KUKA KRL program: EPS_2_25694_RR04_A_20260114065914.src

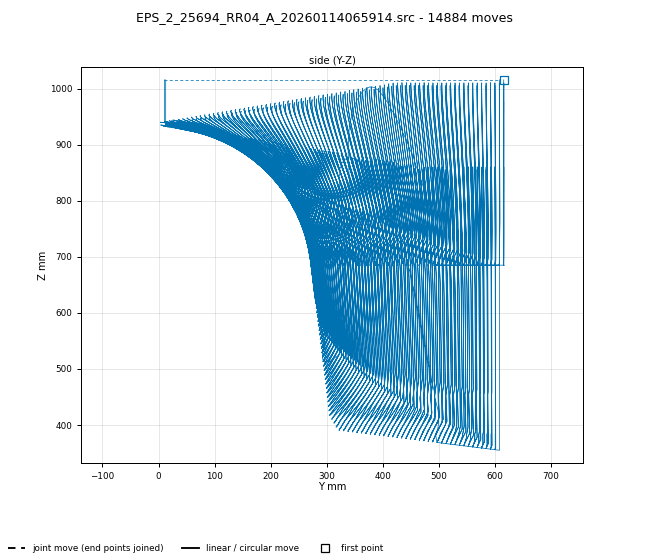
[picture p0: tool path of EPS_2_25694_RR04_A_20260114065914.src, 14884 of 14886 moves have a stored position in this frame; points joined in program order, loops and branches not executed]
&ACCESS RVP
&REL 4
&COMMENT QRS 19112012
&PARAM EDITMASK = *
DEF PART()
EXT BAS (BAS_COMMAND :IN,REAL :IN )
INT I
BAS (#INITMOV,0 )

;KUKA QRS Post kuka4.cps  Date:22-06-2017 !

File_ID=2965

QRS_PRE_INIT()

;Init var - Until changes are made in qrs_pre_init
Outlet_Square_prg=0
Inlet_1_Square_prg=0
Inlet_2_Square_prg=0
Inlet_3_Square_prg=0
Inlet_4_Square_prg=0
Inlet_5_Square_prg=0

Outlet_1={X 0.000, Y 425.000, Z 739.000, B 0.000, E1 0.000 }
Inlet_1={X 0.000, Y 466.000, Z 567.000, B 0.000, E1 180.000 }
Outlet_1_type=533
Inlet_1_type=457
;QRS#1=Sidecore dimensions
;QRS#2=525-21" Concrete
;QRS#3=450-18" Concrete
;QRS#4=
;QRS#5=
;QRS#6=
;QRS#7=
;QRS#8=
;QRS#9=S306-32
;QRS#10=28A PSX-2
;QRS#11=
;QRS#12=
;QRS#13=
;QRS#14=
;QRS#15=
;QRS#16=1220x127x1372 4,5'
;QRS#17=EPS Height
;QRS#18=1005,5
;QRS#19=*
;QRS#20= UPDATED VERSION 22-06-2017
;QRS#21=*
Outlet_Square=0250
Inlet_1_Square=0250
Inlet_2_Square=0
Inlet_3_Square=0
Inlet_4_Square=0
Inlet_5_Square=0
Mill_Square=1
Outlet_Square_Prg=263
Inlet_1_Square_prg=274

QRS_INIT()

$ADVANCE=5

; T1
PTP {E1 172.545,E2 172.545}
PTP {X 0,Y 615.546,A -85,B 0,C 180,E1 172.545,E2 172.545,E3 0,E4 0,E5 0,E6 0}
QRS_SPEED_INIT()
LIN {X 0,Y 615.546,Z 1015.5,A -85,B 0,C 180,E1 172.545,E2 172.545,E3 0,E4 0,E5 0,E6 0} C_VEL
LIN {X 0,Y 615.546,Z 687.03,A -85,B 0,C 180,E1 172.545,E2 172.545} C_VEL
LIN {X 0,Y 615.492,Z 685.03,A -85,B 0,C 180,E1 172.731,E2 172.731} C_VEL
LIN {X 0,Y 615.811,Z 685.03,A -85,B 0,C 180,E1 176.52,E2 176.52} C_VEL
LIN {X 0,Y 615.861,Z 685.03,A -85,B 0,C 180,E1 181.159,E2 181.159} C_VEL
LIN {X 0,Y 615.796,Z 685.03,A -85,B 0,C 180,E1 185.807,E2 185.807} C_VEL
LIN {X 0,Y 615.764,Z 685.03,A -85,B 0,C 180,E1 190.494,E2 190.494} C_VEL
LIN {X 0,Y 615.78,Z 685.03,A -85,B 0,C 180,E1 195.253,E2 195.253} C_VEL
LIN {X 0,Y 615.726,Z 685.03,A -85,B 0,C 180,E1 200.124,E2 200.124} C_VEL
LIN {X 0,Y 615.726,Z 685.03,A -85,B 0,C 180,E1 205.151,E2 205.151} C_VEL
LIN {X 0,Y 615.183,Z 685.03,A -85,B 0,C 180,E1 207.768,E2 207.768} C_VEL
LIN {X 0,Y 615.676,Z 685.03,A -85,B 0,C 180,E1 210.398,E2 210.398} C_VEL
LIN {X 0,Y 615.111,Z 685.03,A -85,B 0,C 180,E1 213.847,E2 213.847} C_VEL
LIN {X 0,Y 615.672,Z 685.03,A -85,B 0,C 180,E1 215.942,E2 215.942} C_VEL
LIN {X 0,Y 615.221,Z 685.03,A -85,B 0,C 180,E1 217.827,E2 217.827} C_VEL
LIN {X 0,Y 615.646,Z 685.03,A -85,B 0,C 180,E1 221.91,E2 221.91} C_VEL
LIN {X 0,Y 615.206,Z 685.03,A -85,B 0,C 180,E1 225.149,E2 225.149} C_VEL
LIN {X 0,Y 615.631,Z 685.03,A -85,B 0,C 180,E1 228.094,E2 228.094} C_VEL
LIN {X 0,Y 615.6,Z 685.03,A -85,B 0,C 180,E1 232.135,E2 232.135} C_VEL
LIN {X 0,Y 615.584,Z 685.03,A -85,B 0,C 180,E1 234.056,E2 234.056} C_VEL
LIN {X 0,Y 615.733,Z 685.03,A -85,B 0,C 180,E1 236.075,E2 236.075} C_VEL
LIN {X 0,Y 615.772,Z 685.03,A -85,B 0,C 180,E1 236.884,E2 236.884} C_VEL
LIN {X 0,Y 615.674,Z 685.03,A -85,B 0,C 180,E1 239.605,E2 239.605} C_VEL
LIN {X 0,Y 615.593,Z 685.03,A -85,B 0,C 180,E1 240.51,E2 240.51} C_VEL
LIN {X 0,Y 615.33,Z 685.03,A -85,B 0,C 180,E1 240.559,E2 240.559} C_VEL
LIN {X 0,Y 615.244,Z 685.519,A -85,B 0,C 180,E1 240.579,E2 240.579} C_VEL
LIN {X 0,Y 615.438,Z 754.445,A -85,B 0,C 180,E1 241.499,E2 241.499} C_VEL
LIN {X 0,Y 615.518,Z 765.253,A -85,B 0,C 180,E1 241.679,E2 241.679} C_VEL
LIN {X 0,Y 615.547,Z 778.462,A -85,B 0,C 180,E1 241.958,E2 241.958} C_VEL
LIN {X 0,Y 615.507,Z 788.764,A -85,B 0,C 180,E1 242.217,E2 242.217} C_VEL
LIN {X 0,Y 615.684,Z 804.589,A -85,B 0,C 180,E1 242.709,E2 242.709} C_VEL
LIN {X 0,Y 615.643,Z 817.012,A -85,B 0,C 180,E1 243.155,E2 243.155} C_VEL
LIN {X 0,Y 615.565,Z 826.929,A -85,B 0,C 180,E1 243.556,E2 243.556} C_VEL
LIN {X 0,Y 615.705,Z 842.642,A -85,B 0,C 180,E1 244.289,E2 244.289} C_VEL
LIN {X 0,Y 615.691,Z 854.976,A -85,B 0,C 180,E1 244.938,E2 244.938} C_VEL
LIN {X 0,Y 615.678,Z 866.612,A -85,B 0,C 180,E1 245.617,E2 245.617} C_VEL
LIN {X 0,Y 615.714,Z 878.42,A -85,B 0,C 180,E1 246.381,E2 246.381} C_VEL
LIN {X 0,Y 615.719,Z 889.111,A -85,B 0,C 180,E1 247.137,E2 247.137} C_VEL
LIN {X 0,Y 615.716,Z 900.416,A -85,B 0,C 180,E1 248.014,E2 248.014} C_VEL
LIN {X 0,Y 615.703,Z 909.675,A -85,B 0,C 180,E1 248.793,E2 248.793} C_VEL
LIN {X 0,Y 615.752,Z 919.81,A -85,B 0,C 180,E1 249.725,E2 249.725} C_VEL
LIN {X 0,Y 615.721,Z 929.071,A -85,B 0,C 180,E1 250.648,E2 250.648} C_VEL
LIN {X 0,Y 615.679,Z 937.431,A -85,B 0,C 180,E1 251.55,E2 251.55} C_VEL
LIN {X 0,Y 615.758,Z 945.789,A -85,B 0,C 180,E1 252.533,E2 252.533} C_VEL
LIN {X 0,Y 615.711,Z 953.693,A -85,B 0,C 180,E1 253.543,E2 253.543} C_VEL
LIN {X 0,Y 615.576,Z 960.436,A -85,B 0,C 180,E1 254.474,E2 254.474} C_VEL
LIN {X 0,Y 615.669,Z 968.069,A -85,B 0,C 180,E1 255.646,E2 255.646} C_VEL
LIN {X 0,Y 615.808,Z 973.445,A -85,B 0,C 180,E1 256.545,E2 256.545} C_VEL
LIN {X 0,Y 615.572,Z 979.916,A -85,B 0,C 180,E1 257.729,E2 257.729} C_VEL
LIN {X 0,Y 615.608,Z 985.63,A -85,B 0,C 180,E1 258.914,E2 258.914} C_VEL
LIN {X 0,Y 615.819,Z 990.639,A -85,B 0,C 180,E1 260.097,E2 260.097} C_VEL
LIN {X 0,Y 615.602,Z 995.067,A -85,B 0,C 180,E1 261.269,E2 261.269} C_VEL
LIN {X 0,Y 615.662,Z 999.448,A -85,B 0,C 180,E1 262.653,E2 262.653} C_VEL
LIN {X 0,Y 615.802,Z 1002.364,A -85,B 0,C 180,E1 263.748,E2 263.748} C_VEL
LIN {X 0,Y 615.545,Z 1005.382,A -85,B 0,C 180,E1 265.123,E2 265.123} C_VEL
LIN {X 0,Y 615.635,Z 1007.593,A -85,B 0,C 180,E1 266.519,E2 266.519} C_VEL
LIN {X 0,Y 615.819,Z 1008.67,A -85,B 0,C 180,E1 267.449,E2 267.449} C_VEL
LIN {X 0,Y 615.544,Z 1009.716,A -85,B 0,C 180,E1 268.84,E2 268.84} C_VEL
LIN {X 0,Y 615.842,Z 1009.659,A -85,B 0,C 180,E1 271.16,E2 271.16} C_VEL
LIN {X 0,Y 615.626,Z 1009.07,A -85,B 0,C 180,E1 272.088,E2 272.088} C_VEL
LIN {X 0,Y 615.536,Z 1007.611,A -85,B 0,C 180,E1 273.482,E2 273.482} C_VEL
LIN {X 0,Y 615.805,Z 1005.333,A -85,B 0,C 180,E1 274.875,E2 274.875} C_VEL
LIN {X 0,Y 615.605,Z 1002.405,A -85,B 0,C 180,E1 276.252,E2 276.252} C_VEL
LIN {X 0,Y 615.625,Z 999.258,A -85,B 0,C 180,E1 277.421,E2 277.421} C_VEL
LIN {X 0,Y 615.798,Z 995.034,A -85,B 0,C 180,E1 278.729,E2 278.729} C_VEL
LIN {X 0,Y 615.583,Z 990.671,A -85,B 0,C 180,E1 279.907,E2 279.907} C_VEL
LIN {X 0,Y 615.638,Z 985.623,A -85,B 0,C 180,E1 281.086,E2 281.086} C_VEL
LIN {X 0,Y 615.808,Z 979.885,A -85,B 0,C 180,E1 282.267,E2 282.267} C_VEL
LIN {X 0,Y 615.627,Z 973.459,A -85,B 0,C 180,E1 283.46,E2 283.46} C_VEL
LIN {X 0,Y 615.697,Z 966.199,A -85,B 0,C 180,E1 284.654,E2 284.654} C_VEL
LIN {X 0,Y 615.81,Z 960.634,A -85,B 0,C 180,E1 285.488,E2 285.488} C_VEL
LIN {X 0,Y 615.662,Z 951.204,A -85,B 0,C 180,E1 286.79,E2 286.79} C_VEL
LIN {X 0,Y 615.736,Z 942.609,A -85,B 0,C 180,E1 287.852,E2 287.852} C_VEL
LIN {X 0,Y 615.77,Z 934.421,A -85,B 0,C 180,E1 288.783,E2 288.783} C_VEL
LIN {X 0,Y 615.695,Z 924.535,A -85,B 0,C 180,E1 289.815,E2 289.815} C_VEL
LIN {X 0,Y 615.712,Z 916.55,A -85,B 0,C 180,E1 290.587,E2 290.587} C_VEL
LIN {X 0,Y 615.743,Z 906.049,A -85,B 0,C 180,E1 291.517,E2 291.517} C_VEL
LIN {X 0,Y 615.702,Z 896.053,A -85,B 0,C 180,E1 292.335,E2 292.335} C_VEL
LIN {X 0,Y 615.701,Z 886.308,A -85,B 0,C 180,E1 293.07,E2 293.07} C_VEL
LIN {X 0,Y 615.683,Z 874.638,A -85,B 0,C 180,E1 293.873,E2 293.873} C_VEL
LIN {X 0,Y 615.697,Z 862.6,A -85,B 0,C 180,E1 294.623,E2 294.623} C_VEL
LIN {X 0,Y 615.65,Z 851.918,A -85,B 0,C 180,E1 295.232,E2 295.232} C_VEL
LIN {X 0,Y 615.643,Z 841.055,A -85,B 0,C 180,E1 295.795,E2 295.795} C_VEL
LIN {X 0,Y 615.699,Z 826.912,A -85,B 0,C 180,E1 296.438,E2 296.438} C_VEL
LIN {X 0,Y 615.612,Z 813.716,A -85,B 0,C 180,E1 296.969,E2 296.969} C_VEL
LIN {X 0,Y 615.55,Z 804.569,A -85,B 0,C 180,E1 297.298,E2 297.298} C_VEL
LIN {X 0,Y 615.613,Z 787.831,A -85,B 0,C 180,E1 297.801,E2 297.801} C_VEL
LIN {X 0,Y 615.471,Z 776.05,A -85,B 0,C 180,E1 298.103,E2 298.103} C_VEL
LIN {X 0,Y 615.643,Z 762.933,A -85,B 0,C 180,E1 298.359,E2 298.359} C_VEL
LIN {X 0,Y 615.608,Z 744.148,A -85,B 0,C 180,E1 298.636,E2 298.636} C_VEL
LIN {X 0,Y 615.246,Z 685.03,A -85,B 0,C 180,E1 299.433,E2 299.433} C_VEL
LIN {X 0,Y 615.499,Z 685.03,A -85,B 0,C 180,E1 299.474,E2 299.474} C_VEL
LIN {X 0,Y 615.685,Z 685.03,A -85,B 0,C 180,E1 300.395,E2 300.395} C_VEL
LIN {X 0,Y 615.866,Z 685.03,A -85,B 0,C 180,E1 303.111,E2 303.111} C_VEL
LIN {X 0,Y 615.556,Z 685.03,A -85,B 0,C 180,E1 305.946,E2 305.946} C_VEL
LIN {X 0,Y 615.615,Z 685.03,A -85,B 0,C 180,E1 307.866,E2 307.866} C_VEL
LIN {X 0,Y 615.631,Z 685.03,A -85,B 0,C 180,E1 311.906,E2 311.906} C_VEL
LIN {X 0,Y 615.209,Z 685.03,A -85,B 0,C 180,E1 315.144,E2 315.144} C_VEL
LIN {X 0,Y 615.686,Z 685.03,A -85,B 0,C 180,E1 318.094,E2 318.094} C_VEL
LIN {X 0,Y 615.541,Z 685.03,A -85,B 0,C 180,E1 322.136,E2 322.136} C_VEL
LIN {X 0,Y 615.511,Z 685.03,A -85,B 0,C 180,E1 324.047,E2 324.047} C_VEL
LIN {X 0,Y 615.673,Z 685.03,A -85,B 0,C 180,E1 326.076,E2 326.076} C_VEL
LIN {X 0,Y 615.675,Z 685.03,A -85,B 0,C 180,E1 326.874,E2 326.874} C_VEL
LIN {X 0,Y 615.495,Z 685.03,A -85,B 0,C 180,E1 330.517,E2 330.517} C_VEL
LIN {X 0,Y 615.462,Z 685.03,A -85,B 0,C 180,E1 332.245,E2 332.245} C_VEL
LIN {X 0,Y 615.386,Z 685.03,A -85,B 0,C 180,E1 335.665,E2 335.665} C_VEL
LIN {X 0,Y 615.551,Z 685.03,A -85,B 0,C 180,E1 337.379,E2 337.379} C_VEL
LIN {X 0,Y 615.774,Z 685.03,A -85,B 0,C 180,E1 341.999,E2 341.999} C_VEL
LIN {X 0,Y 615.786,Z 685.03,A -85,B 0,C 180,E1 342.329,E2 342.329} C_VEL
LIN {X 0,Y 615.756,Z 685.03,A -85,B 0,C 180,E1 347.137,E2 347.137} C_VEL
LIN {X 0,Y 615.771,Z 685.03,A -85,B 0,C 180,E1 351.856,E2 351.856} C_VEL
LIN {X 0,Y 615.848,Z 685.03,A -85,B 0,C 180,E1 356.52,E2 356.52} C_VEL
LIN {X 0,Y 615.86,Z 685.03,A -85,B 0,C 180,E1 361.159,E2 361.159} C_VEL
LIN {X 0,Y 615.803,Z 685.03,A -85,B 0,C 180,E1 365.807,E2 365.807} C_VEL
LIN {X 0,Y 615.789,Z 685.03,A -85,B 0,C 180,E1 370.494,E2 370.494} C_VEL
LIN {X 0,Y 615.809,Z 685.03,A -85,B 0,C 180,E1 375.252,E2 375.252} C_VEL
LIN {X 0,Y 615.742,Z 685.03,A -85,B 0,C 180,E1 380.124,E2 380.124} C_VEL
LIN {X 0,Y 615.764,Z 685.03,A -85,B 0,C 180,E1 385.15,E2 385.15} C_VEL
LIN {X 0,Y 615.376,Z 685.03,A -85,B 0,C 180,E1 389.463,E2 389.463} C_VEL
LIN {X 0,Y 615.696,Z 685.03,A -85,B 0,C 180,E1 390.397,E2 390.397} C_VEL
LIN {X 0,Y 615.123,Z 685.03,A -85,B 0,C 180,E1 393.848,E2 393.848} C_VEL
LIN {X 0,Y 615.679,Z 685.03,A -85,B 0,C 180,E1 395.942,E2 395.942} C_VEL
LIN {X 0,Y 615.41,Z 685.03,A -85,B 0,C 180,E1 397.848,E2 397.848} C_VEL
LIN {X 0,Y 615.356,Z 685.03,A -85,B 0,C 180,E1 398.886,E2 398.886} C_VEL
LIN {X 0,Y 615.631,Z 685.03,A -85,B 0,C 180,E1 401.507,E2 401.507} C_VEL
LIN {X 0,Y 615.653,Z 685.03,A -85,B 0,C 180,E1 405.107,E2 405.107} C_VEL
LIN {X 0,Y 615.249,Z 685.03,A -85,B 0,C 180,E1 408.539,E2 408.539} C_VEL
LIN {X 0,Y 615.649,Z 685.03,A -85,B 0,C 180,E1 411.14,E2 411.14} C_VEL
LIN {X 0,Y 615.653,Z 685.03,A -85,B 0,C 180,E1 416.086,E2 416.086} C_VEL
LIN {X 0,Y 615.746,Z 685.03,A -85,B 0,C 180,E1 416.881,E2 416.881} C_VEL
LIN {X 0,Y 615.563,Z 685.03,A -85,B 0,C 180,E1 420.515,E2 420.515} C_VEL
LIN {X 0,Y 615.554,Z 685.03,A -85,B 0,C 180,E1 422.252,E2 422.252} C_VEL
LIN {X 0,Y 615.586,Z 685.03,A -85,B 0,C 180,E1 425.635,E2 425.635} C_VEL
LIN {X 0,Y 615.626,Z 685.03,A -85,B 0,C 180,E1 426.524,E2 426.524} C_VEL
LIN {X 0,Y 615.741,Z 696.131,A -85,B 0,C 180,E1 426.945,E2 426.945} C_VEL
LIN {X 0,Y 615.761,Z 704.206,A -85,B 0,C 180,E1 427.278,E2 427.278} C_VEL
LIN {X 0,Y 615.706,Z 714.196,A -85,B 0,C 180,E1 427.733,E2 427.733} C_VEL
LIN {X 0,Y 615.726,Z 725.668,A -85,B 0,C 180,E1 428.326,E2 428.326} C_VEL
LIN {X 0,Y 615.756,Z 736.464,A -85,B 0,C 180,E1 428.95,E2 428.95} C_VEL
LIN {X 0,Y 615.75,Z 746.203,A -85,B 0,C 180,E1 429.569,E2 429.569} C_VEL
LIN {X 0,Y 615.753,Z 755.081,A -85,B 0,C 180,E1 430.187,E2 430.187} C_VEL
LIN {X 0,Y 615.748,Z 765.126,A -85,B 0,C 180,E1 430.955,E2 430.955} C_VEL
LIN {X 0,Y 615.773,Z 773.255,A -85,B 0,C 180,E1 431.632,E2 431.632} C_VEL
LIN {X 0,Y 615.741,Z 782.057,A -85,B 0,C 180,E1 432.43,E2 432.43} C_VEL
LIN {X 0,Y 615.697,Z 789.212,A -85,B 0,C 180,E1 433.131,E2 433.131} C_VEL
LIN {X 0,Y 615.74,Z 797.147,A -85,B 0,C 180,E1 433.981,E2 433.981} C_VEL
LIN {X 0,Y 615.809,Z 803.754,A -85,B 0,C 180,E1 434.749,E2 434.749} C_VEL
LIN {X 0,Y 615.685,Z 810.869,A -85,B 0,C 180,E1 435.646,E2 435.646} C_VEL
LIN {X 0,Y 615.683,Z 817.337,A -85,B 0,C 180,E1 436.541,E2 436.541} C_VEL
LIN {X 0,Y 615.817,Z 823.206,A -85,B 0,C 180,E1 437.437,E2 437.437} C_VEL
LIN {X 0,Y 615.707,Z 828.568,A -85,B 0,C 180,E1 438.324,E2 438.324} C_VEL
LIN {X 0,Y 615.629,Z 834.87,A -85,B 0,C 180,E1 439.504,E2 439.504} C_VEL
LIN {X 0,Y 615.74,Z 839.094,A -85,B 0,C 180,E1 440.389,E2 440.389} C_VEL
LIN {X 0,Y 615.768,Z 842.865,A -85,B 0,C 180,E1 441.271,E2 441.271} C_VEL
LIN {X 0,Y 615.623,Z 847.726,A -85,B 0,C 180,E1 442.579,E2 442.579} C_VEL
LIN {X 0,Y 615.757,Z 851.304,A -85,B 0,C 180,E1 443.75,E2 443.75} C_VEL
LIN {X 0,Y 615.736,Z 853.695,A -85,B 0,C 180,E1 444.658,E2 444.658} C_VEL
LIN {X 0,Y 615.634,Z 856.541,A -85,B 0,C 180,E1 446.054,E2 446.054} C_VEL
LIN {X 0,Y 615.679,Z 857.314,A -85,B 0,C 180,E1 446.519,E2 446.519} C_VEL
LIN {X 0,Y 615.827,Z 858.489,A -85,B 0,C 180,E1 447.448,E2 447.448} C_VEL
LIN {X 0,Y 615.722,Z 859.014,A -85,B 0,C 180,E1 447.912,E2 447.912} C_VEL
LIN {X 0,Y 615.59,Z 859.697,A -85,B 0,C 180,E1 448.84,E2 448.84} C_VEL
LIN {X 0,Y 615.619,Z 859.93,A -85,B 0,C 180,E1 449.768,E2 449.768} C_VEL
LIN {X 0,Y 615.785,Z 859.595,A -85,B 0,C 180,E1 451.159,E2 451.159} C_VEL
LIN {X 0,Y 615.595,Z 858.426,A -85,B 0,C 180,E1 452.552,E2 452.552} C_VEL
LIN {X 0,Y 615.657,Z 857.167,A -85,B 0,C 180,E1 453.481,E2 453.481} C_VEL
LIN {X 0,Y 615.748,Z 856.37,A -85,B 0,C 180,E1 453.945,E2 453.945} C_VEL
LIN {X 0,Y 615.735,Z 854.511,A -85,B 0,C 180,E1 454.875,E2 454.875} C_VEL
LIN {X 0,Y 615.653,Z 853.513,A -85,B 0,C 180,E1 455.342,E2 455.342} C_VEL
LIN {X 0,Y 615.602,Z 849.864,A -85,B 0,C 180,E1 456.665,E2 456.665} C_VEL
LIN {X 0,Y 615.761,Z 847.084,A -85,B 0,C 180,E1 457.52,E2 457.52} C_VEL
LIN {X 0,Y 615.802,Z 844.751,A -85,B 0,C 180,E1 458.142,E2 458.142} C_VEL
LIN {X 0,Y 615.65,Z 841.238,A -85,B 0,C 180,E1 459.024,E2 459.024} C_VEL
LIN {X 0,Y 615.622,Z 838.719,A -85,B 0,C 180,E1 459.612,E2 459.612} C_VEL
LIN {X 0,Y 615.757,Z 832.894,A -85,B 0,C 180,E1 460.788,E2 460.788} C_VEL
LIN {X 0,Y 615.749,Z 828.046,A -85,B 0,C 180,E1 461.675,E2 461.675} C_VEL
LIN {X 0,Y 615.66,Z 822.681,A -85,B 0,C 180,E1 462.566,E2 462.566} C_VEL
LIN {X 0,Y 615.742,Z 815.692,A -85,B 0,C 180,E1 463.606,E2 463.606} C_VEL
LIN {X 0,Y 615.788,Z 809.065,A -85,B 0,C 180,E1 464.501,E2 464.501} C_VEL
LIN {X 0,Y 615.684,Z 800.716,A -85,B 0,C 180,E1 465.523,E2 465.523} C_VEL
LIN {X 0,Y 615.718,Z 793.726,A -85,B 0,C 180,E1 466.306,E2 466.306} C_VEL
LIN {X 0,Y 615.785,Z 785.347,A -85,B 0,C 180,E1 467.162,E2 467.162} C_VEL
LIN {X 0,Y 615.744,Z 777.922,A -85,B 0,C 180,E1 467.865,E2 467.865} C_VEL
LIN {X 0,Y 615.74,Z 769.905,A -85,B 0,C 180,E1 468.566,E2 468.566} C_VEL
LIN {X 0,Y 615.748,Z 760.061,A -85,B 0,C 180,E1 469.351,E2 469.351} C_VEL
LIN {X 0,Y 615.758,Z 750.554,A -85,B 0,C 180,E1 470.044,E2 470.044} C_VEL
LIN {X 0,Y 615.741,Z 741.275,A -85,B 0,C 180,E1 470.662,E2 470.662} C_VEL
LIN {X 0,Y 615.705,Z 731.012,A -85,B 0,C 180,E1 471.285,E2 471.285} C_VEL
LIN {X 0,Y 615.735,Z 721.063,A -85,B 0,C 180,E1 471.829,E2 471.829} C_VEL
LIN {X 0,Y 615.723,Z 710.661,A -85,B 0,C 180,E1 472.343,E2 472.343} C_VEL
LIN {X 0,Y 615.656,Z 699.442,A -85,B 0,C 180,E1 472.837,E2 472.837} C_VEL
LIN {X 0,Y 615.443,Z 689.43,A -85,B 0,C 180,E1 473.235,E2 473.235} C_VEL
LIN {X 0,Y 615.249,Z 685.03,A -85,B 0,C 180,E1 473.397,E2 473.397} C_VEL
LIN {X 0,Y 615.705,Z 685.03,A -85,B 0,C 180,E1 473.504,E2 473.504} C_VEL
LIN {X 0,Y 615.521,Z 685.03,A -85,B 0,C 180,E1 474.765,E2 474.765} C_VEL
LIN {X 0,Y 615.766,Z 685.03,A -85,B 0,C 180,E1 477.736,E2 477.736} C_VEL
LIN {X 0,Y 615.191,Z 685.03,A -85,B 0,C 180,E1 480.421,E2 480.421} C_VEL
LIN {X 0,Y 615.731,Z 685.03,A -85,B 0,C 180,E1 483.119,E2 483.119} C_VEL
LIN {X 0,Y 615.647,Z 685.03,A -85,B 0,C 180,E1 483.913,E2 483.913} C_VEL
LIN {X 0,Y 615.65,Z 685.03,A -85,B 0,C 180,E1 488.859,E2 488.859} C_VEL
LIN {X 0,Y 615.238,Z 685.03,A -85,B 0,C 180,E1 491.938,E2 491.938} C_VEL
LIN {X 0,Y 615.647,Z 685.03,A -85,B 0,C 180,E1 494.892,E2 494.892} C_VEL
LIN {X 0,Y 615.63,Z 685.03,A -85,B 0,C 180,E1 498.492,E2 498.492} C_VEL
LIN {X 0,Y 615.363,Z 685.03,A -85,B 0,C 180,E1 501.115,E2 501.115} C_VEL
LIN {X 0,Y 615.412,Z 685.03,A -85,B 0,C 180,E1 502.15,E2 502.15} C_VEL
LIN {X 0,Y 615.688,Z 685.03,A -85,B 0,C 180,E1 504.059,E2 504.059} C_VEL
LIN {X 0,Y 615.124,Z 685.03,A -85,B 0,C 180,E1 506.84,E2 506.84} C_VEL
LIN {X 0,Y 615.697,Z 685.03,A -85,B 0,C 180,E1 509.603,E2 509.603} C_VEL
LIN {X 0,Y 615.213,Z 685.03,A -85,B 0,C 180,E1 512.233,E2 512.233} C_VEL
LIN {X 0,Y 615.762,Z 685.03,A -85,B 0,C 180,E1 514.85,E2 514.85} C_VEL
LIN {X 0,Y 615.747,Z 685.03,A -85,B 0,C 180,E1 519.877,E2 519.877} C_VEL
LIN {X 0,Y 615.473,Z 685.03,A -85,B 0,C 180,E1 522.32,E2 522.32} C_VEL
LIN {X 0,Y 615.601,Z 685.03,A -85,B 0,C 180,E1 524.743,E2 524.743} C_VEL
LIN {X 0,Y 615.815,Z 685.03,A -85,B 0,C 180,E1 527.139,E2 527.139} C_VEL
LIN {X 0,Y 615.786,Z 685.03,A -85,B 0,C 180,E1 531.856,E2 531.856} C_VEL
LIN {X 0,Y 615.492,Z 685.03,A -85,B 0,C 180,E1 532.731,E2 532.731} C_VEL
LIN {X 0,Y 611.488,Z 685.03,A -85,B 0,C 180,E1 534.318,E2 534.318} C_VEL
LIN {X 0,Y 607.633,Z 685.03,A -85,B 0,C 180,E1 535.926,E2 535.926} C_VEL
LIN {X 0,Y 607.869,Z 685.03,A -85,B 0,C 180,E1 541.425,E2 541.425} C_VEL
LIN {X 0,Y 607.617,Z 685.03,A -85,B 0,C 180,E1 546.595,E2 546.595} C_VEL
LIN {X 0,Y 607.525,Z 685.03,A -85,B 0,C 180,E1 551.463,E2 551.463} C_VEL
LIN {X 0,Y 607.629,Z 685.03,A -85,B 0,C 180,E1 555.855,E2 555.855} C_VEL
LIN {X 0,Y 607.738,Z 685.03,A -85,B 0,C 180,E1 560.343,E2 560.343} C_VEL
LIN {X 0,Y 607.749,Z 685.03,A -85,B 0,C 180,E1 564.968,E2 564.968} C_VEL
LIN {X 0,Y 607.546,Z 685.03,A -85,B 0,C 180,E1 569.786,E2 569.786} C_VEL
LIN {X 0,Y 607.544,Z 685.03,A -85,B 0,C 180,E1 576.592,E2 576.592} C_VEL
LIN {X 0,Y 607.666,Z 685.03,A -85,B 0,C 180,E1 582.104,E2 582.104} C_VEL
LIN {X 0,Y 607.705,Z 685.03,A -85,B 0,C 180,E1 588.152,E2 588.152} C_VEL
LIN {X 0,Y 607.619,Z 685.03,A -85,B 0,C 180,E1 593.414,E2 593.414} C_VEL
LIN {X 0,Y 607.66,Z 685.03,A -85,B 0,C 180,E1 598.568,E2 598.568} C_VEL
LIN {X 0,Y 607.716,Z 685.03,A -85,B 0,C 180,E1 600.166,E2 600.166} C_VEL
LIN {X 0,Y 608.571,Z 773.176,A -85,B 0,C 180,E1 601.49,E2 601.49} C_VEL
LIN {X 0,Y 608.554,Z 810.788,A -85,B 0,C 180,E1 602.586,E2 602.586} C_VEL
LIN {X 0,Y 608.43,Z 846.811,A -85,B 0,C 180,E1 604.178,E2 604.178} C_VEL
LIN {X 0,Y 608.276,Z 881.947,A -85,B 0,C 180,E1 606.323,E2 606.323} C_VEL
LIN {X 0,Y 608.109,Z 914.005,A -85,B 0,C 180,E1 608.911,E2 608.911} C_VEL
LIN {X 0,Y 607.968,Z 942.725,A -85,B 0,C 180,E1 611.926,E2 611.926} C_VEL
LIN {X 0,Y 607.834,Z 967.192,A -85,B 0,C 180,E1 615.295,E2 615.295} C_VEL
LIN {X 0,Y 607.754,Z 986.44,A -85,B 0,C 180,E1 618.906,E2 618.906} C_VEL
LIN {X 0,Y 607.787,Z 999.718,A -85,B 0,C 180,E1 622.51,E2 622.51} C_VEL
LIN {X 0,Y 607.67,Z 1006.956,A -85,B 0,C 180,E1 625.728,E2 625.728} C_VEL
LIN {X 0,Y 607.699,Z 1010.086,A -85,B 0,C 180,E1 628.577,E2 628.577} C_VEL
LIN {X 0,Y 607.888,Z 1010.086,A -85,B 0,C 180,E1 631.422,E2 631.422} C_VEL
LIN {X 0,Y 607.905,Z 1005.757,A -85,B 0,C 180,E1 634.984,E2 634.984} C_VEL
LIN {X 0,Y 607.891,Z 995.073,A -85,B 0,C 180,E1 638.925,E2 638.925} C_VEL
LIN {X 0,Y 607.907,Z 979.451,A -85,B 0,C 180,E1 642.545,E2 642.545} C_VEL
LIN {X 0,Y 607.956,Z 958.35,A -85,B 0,C 180,E1 646.029,E2 646.029} C_VEL
LIN {X 0,Y 608.033,Z 932.207,A -85,B 0,C 180,E1 649.269,E2 649.269} C_VEL
LIN {X 0,Y 608.169,Z 902.026,A -85,B 0,C 180,E1 652.138,E2 652.138} C_VEL
LIN {X 0,Y 608.316,Z 868.893,A -85,B 0,C 180,E1 654.551,E2 654.551} C_VEL
LIN {X 0,Y 608.479,Z 832.749,A -85,B 0,C 180,E1 656.512,E2 656.512} C_VEL
LIN {X 0,Y 608.583,Z 795.987,A -85,B 0,C 180,E1 657.91,E2 657.91} C_VEL
LIN {X 0,Y 608.707,Z 760.135,A -85,B 0,C 180,E1 658.756,E2 658.756} C_VEL
LIN {X 0,Y 607.685,Z 685.523,A -85,B 0,C 180,E1 659.824,E2 659.824} C_VEL
LIN {X 0,Y 607.985,Z 685.03,A -85,B 0,C 180,E1 663.095,E2 663.095} C_VEL
LIN {X 0,Y 607.56,Z 685.03,A -85,B 0,C 180,E1 668.384,E2 668.384} C_VEL
LIN {X 0,Y 607.653,Z 685.03,A -85,B 0,C 180,E1 672.105,E2 672.105} C_VEL
LIN {X 0,Y 607.776,Z 685.03,A -85,B 0,C 180,E1 678.146,E2 678.146} C_VEL
LIN {X 0,Y 607.571,Z 685.03,A -85,B 0,C 180,E1 683.41,E2 683.41} C_VEL
LIN {X 0,Y 607.535,Z 685.03,A -85,B 0,C 180,E1 687.617,E2 687.617} C_VEL
LIN {X 0,Y 607.541,Z 685.03,A -85,B 0,C 180,E1 691.84,E2 691.84} C_VEL
LIN {X 0,Y 607.426,Z 685.03,A -85,B 0,C 180,E1 698.12,E2 698.12} C_VEL
LIN {X 0,Y 607.762,Z 685.03,A -85,B 0,C 180,E1 702.664,E2 702.664} C_VEL
LIN {X 0,Y 607.828,Z 685.03,A -85,B 0,C 180,E1 707.087,E2 707.087} C_VEL
LIN {X 0,Y 607.541,Z 685.03,A -85,B 0,C 180,E1 712.864,E2 712.864} C_VEL
LIN {X 0,Y 607.724,Z 685.03,A -85,B 0,C 180,E1 717.151,E2 717.151} C_VEL
LIN {X 0,Y 607.851,Z 685.03,A -85,B 0,C 180,E1 721.42,E2 721.42} C_VEL
LIN {X 0,Y 607.621,Z 685.03,A -85,B 0,C 180,E1 726.598,E2 726.598} C_VEL
LIN {X 0,Y 607.568,Z 685.03,A -85,B 0,C 180,E1 731.457,E2 731.457} C_VEL
LIN {X 0,Y 607.676,Z 685.03,A -85,B 0,C 180,E1 735.848,E2 735.848} C_VEL
LIN {X 0,Y 607.75,Z 685.03,A -85,B 0,C 180,E1 740.337,E2 740.337} C_VEL
LIN {X 0,Y 607.795,Z 685.03,A -85,B 0,C 180,E1 744.96,E2 744.96} C_VEL
LIN {X 0,Y 607.579,Z 685.03,A -85,B 0,C 180,E1 749.778,E2 749.778} C_VEL
LIN {X 0,Y 607.632,Z 685.03,A -85,B 0,C 180,E1 756.579,E2 756.579} C_VEL
LIN {X 0,Y 607.565,Z 685.03,A -85,B 0,C 180,E1 762.105,E2 762.105} C_VEL
LIN {X 0,Y 607.271,Z 685.03,A -85,B 0,C 180,E1 767.862,E2 767.862} C_VEL
LIN {X 0,Y 607.292,Z 685.03,A -85,B 0,C 180,E1 772.658,E2 772.658} C_VEL
LIN {X 0,Y 607.621,Z 685.03,A -85,B 0,C 180,E1 777.593,E2 777.593} C_VEL
LIN {X 0,Y 607.621,Z 685.03,A -85,B 0,C 180,E1 781.845,E2 781.845} C_VEL
LIN {X 0,Y 607.699,Z 685.03,A -85,B 0,C 180,E1 786.198,E2 786.198} C_VEL
LIN {X 0,Y 608.305,Z 720.517,A -85,B 0,C 180,E1 787.772,E2 787.772} C_VEL
LIN {X 0,Y 608.187,Z 753.546,A -85,B 0,C 180,E1 789.815,E2 789.815} C_VEL
LIN {X 0,Y 608.031,Z 783.088,A -85,B 0,C 180,E1 792.301,E2 792.301} C_VEL
LIN {X 0,Y 607.947,Z 808.121,A -85,B 0,C 180,E1 795.093,E2 795.093} C_VEL
LIN {X 0,Y 607.889,Z 828.8,A -85,B 0,C 180,E1 798.183,E2 798.183} C_VEL
LIN {X 0,Y 607.884,Z 844.272,A -85,B 0,C 180,E1 801.434,E2 801.434} C_VEL
LIN {X 0,Y 607.814,Z 855.085,A -85,B 0,C 180,E1 805.015,E2 805.015} C_VEL
LIN {X 0,Y 607.747,Z 860.042,A -85,B 0,C 180,E1 808.577,E2 808.577} C_VEL
LIN {X 0,Y 607.851,Z 859.979,A -85,B 0,C 180,E1 811.423,E2 811.423} C_VEL
LIN {X 0,Y 607.849,Z 854.89,A -85,B 0,C 180,E1 814.985,E2 814.985} C_VEL
LIN {X 0,Y 607.864,Z 843.938,A -85,B 0,C 180,E1 818.566,E2 818.566} C_VEL
LIN {X 0,Y 607.887,Z 827.186,A -85,B 0,C 180,E1 821.999,E2 821.999} C_VEL
LIN {X 0,Y 607.936,Z 805.583,A -85,B 0,C 180,E1 825.137,E2 825.137} C_VEL
LIN {X 0,Y 608.071,Z 779.27,A -85,B 0,C 180,E1 827.978,E2 827.978} C_VEL
LIN {X 0,Y 608.212,Z 748.878,A -85,B 0,C 180,E1 830.42,E2 830.42} C_VEL
LIN {X 0,Y 608.319,Z 715.008,A -85,B 0,C 180,E1 832.42,E2 832.42} C_VEL
LIN {X 0,Y 607.75,Z 685.03,A -85,B 0,C 180,E1 833.751,E2 833.751} C_VEL
LIN {X 0,Y 607.693,Z 685.03,A -85,B 0,C 180,E1 838.151,E2 838.151} C_VEL
LIN {X 0,Y 607.828,Z 685.03,A -85,B 0,C 180,E1 843.105,E2 843.105} C_VEL
LIN {X 0,Y 607.494,Z 685.03,A -85,B 0,C 180,E1 849.653,E2 849.653} C_VEL
LIN {X 0,Y 607.495,Z 685.03,A -85,B 0,C 180,E1 855.94,E2 855.94} C_VEL
LIN {X 0,Y 607.408,Z 685.03,A -85,B 0,C 180,E1 860.366,E2 860.366} C_VEL
LIN {X 0,Y 607.408,Z 685.03,A -85,B 0,C 180,E1 865.159,E2 865.159} C_VEL
LIN {X 0,Y 607.533,Z 685.03,A -85,B 0,C 180,E1 870.381,E2 870.381} C_VEL
LIN {X 0,Y 607.78,Z 685.03,A -85,B 0,C 180,E1 875.039,E2 875.039} C_VEL
LIN {X 0,Y 607.577,Z 685.03,A -85,B 0,C 180,E1 881.168,E2 881.168} C_VEL
LIN {X 0,Y 607.917,Z 685.03,A -85,B 0,C 180,E1 887.095,E2 887.095} C_VEL
LIN {X 0,Y 607.576,Z 685.03,A -85,B 0,C 180,E1 892.87,E2 892.87} C_VEL
LIN {X 0,Y 607.633,Z 685.03,A -85,B 0,C 180,E1 895.926,E2 895.926} C_VEL
LIN {X 0,Y 606.312,Z 685.03,A -85,B 0,C 180,E1 896.74,E2 896.74} C_VEL
LIN {X 0,Y 599.637,Z 685.03,A -85,B 0,C 180,E1 898.951,E2 898.951} C_VEL
LIN {X 0,Y 599.56,Z 685.03,A -85,B 0,C 180,E1 899.16,E2 899.16} C_VEL
LIN {X 0,Y 599.609,Z 685.03,A -85,B 0,C 180,E1 902.888,E2 902.888} C_VEL
LIN {X 0,Y 599.568,Z 685.03,A -85,B 0,C 180,E1 907.232,E2 907.232} C_VEL
LIN {X 0,Y 599.593,Z 685.03,A -85,B 0,C 180,E1 911.617,E2 911.617} C_VEL
LIN {X 0,Y 599.658,Z 685.03,A -85,B 0,C 180,E1 916.071,E2 916.071} C_VEL
LIN {X 0,Y 599.517,Z 685.03,A -85,B 0,C 180,E1 921.363,E2 921.363} C_VEL
LIN {X 0,Y 599.759,Z 685.03,A -85,B 0,C 180,E1 925.324,E2 925.324} C_VEL
LIN {X 0,Y 599.474,Z 685.03,A -85,B 0,C 180,E1 931.147,E2 931.147} C_VEL
LIN {X 0,Y 599.528,Z 685.03,A -85,B 0,C 180,E1 937.162,E2 937.162} C_VEL
LIN {X 0,Y 599.455,Z 685.03,A -85,B 0,C 180,E1 943.113,E2 943.113} C_VEL
LIN {X 0,Y 599.55,Z 685.03,A -85,B 0,C 180,E1 949.127,E2 949.127} C_VEL
LIN {X 0,Y 599.716,Z 685.03,A -85,B 0,C 180,E1 954.639,E2 954.639} C_VEL
LIN {X 0,Y 599.906,Z 685.729,A -85,B 0,C 180,E1 959.752,E2 959.752} C_VEL
LIN {X 0,Y 601.524,Z 693.003,A -85,B 0,C 180,E1 959.94,E2 959.94} C_VEL
LIN {X 0,Y 601.623,Z 773.216,A -85,B 0,C 180,E1 961.131,E2 961.131} C_VEL
LIN {X 0,Y 601.477,Z 809.645,A -85,B 0,C 180,E1 962.194,E2 962.194} C_VEL
LIN {X 0,Y 601.209,Z 844.95,A -85,B 0,C 180,E1 963.745,E2 963.745} C_VEL
LIN {X 0,Y 600.863,Z 880.578,A -85,B 0,C 180,E1 965.915,E2 965.915} C_VEL
LIN {X 0,Y 600.54,Z 913.063,A -85,B 0,C 180,E1 968.545,E2 968.545} C_VEL
LIN {X 0,Y 600.233,Z 941.122,A -85,B 0,C 180,E1 971.495,E2 971.495} C_VEL
LIN {X 0,Y 599.991,Z 965.753,A -85,B 0,C 180,E1 974.875,E2 974.875} C_VEL
LIN {X 0,Y 599.867,Z 984.767,A -85,B 0,C 180,E1 978.39,E2 978.39} C_VEL
LIN {X 0,Y 599.858,Z 997.447,A -85,B 0,C 180,E1 981.683,E2 981.683} C_VEL
LIN {X 0,Y 599.791,Z 1005.757,A -85,B 0,C 180,E1 984.948,E2 984.948} C_VEL
LIN {X 0,Y 599.8,Z 1010.086,A -85,B 0,C 180,E1 988.558,E2 988.558} C_VEL
LIN {X 0,Y 599.981,Z 1010.086,A -85,B 0,C 180,E1 991.441,E2 991.441} C_VEL
LIN {X 0,Y 599.992,Z 1005.757,A -85,B 0,C 180,E1 995.05,E2 995.05} C_VEL
LIN {X 0,Y 599.989,Z 995.073,A -85,B 0,C 180,E1 999.044,E2 999.044} C_VEL
LIN {X 0,Y 600.042,Z 979.452,A -85,B 0,C 180,E1 1002.712,E2 1002.712} C_VEL
LIN {X 0,Y 600.116,Z 957.718,A -85,B 0,C 180,E1 1006.334,E2 1006.334} C_VEL
LIN {X 0,Y 600.342,Z 932.043,A -85,B 0,C 180,E1 1009.544,E2 1009.544} C_VEL
LIN {X 0,Y 600.636,Z 901.457,A -85,B 0,C 180,E1 1012.479,E2 1012.479} C_VEL
LIN {X 0,Y 601.004,Z 866.909,A -85,B 0,C 180,E1 1015,E2 1015} C_VEL
LIN {X 0,Y 601.364,Z 828.855,A -85,B 0,C 180,E1 1017.036,E2 1017.036} C_VEL
LIN {X 0,Y 601.578,Z 789.555,A -85,B 0,C 180,E1 1018.463,E2 1018.463} C_VEL
LIN {X 0,Y 601.799,Z 747.737,A -85,B 0,C 180,E1 1019.308,E2 1019.308} C_VEL
LIN {X 0,Y 600.925,Z 688.986,A -85,B 0,C 180,E1 1020.147,E2 1020.147} C_VEL
LIN {X 0,Y 599.871,Z 685.03,A -85,B 0,C 180,E1 1020.33,E2 1020.33} C_VEL
LIN {X 0,Y 599.676,Z 685.03,A -85,B 0,C 180,E1 1025.363,E2 1025.363} C_VEL
LIN {X 0,Y 599.578,Z 685.03,A -85,B 0,C 180,E1 1030.973,E2 1030.973} C_VEL
LIN {X 0,Y 599.585,Z 685.03,A -85,B 0,C 180,E1 1037.194,E2 1037.194} C_VEL
LIN {X 0,Y 599.667,Z 685.03,A -85,B 0,C 180,E1 1042.848,E2 1042.848} C_VEL
LIN {X 0,Y 599.546,Z 685.03,A -85,B 0,C 180,E1 1048.092,E2 1048.092} C_VEL
LIN {X 0,Y 599.407,Z 685.03,A -85,B 0,C 180,E1 1053.053,E2 1053.053} C_VEL
LIN {X 0,Y 599.531,Z 685.03,A -85,B 0,C 180,E1 1057.817,E2 1057.817} C_VEL
LIN {X 0,Y 599.771,Z 685.03,A -85,B 0,C 180,E1 1062.952,E2 1062.952} C_VEL
LIN {X 0,Y 599.583,Z 685.03,A -85,B 0,C 180,E1 1068.383,E2 1068.383} C_VEL
LIN {X 0,Y 599.64,Z 685.03,A -85,B 0,C 180,E1 1072.769,E2 1072.769} C_VEL
LIN {X 0,Y 599.834,Z 685.03,A -85,B 0,C 180,E1 1077.113,E2 1077.113} C_VEL
LIN {X 0,Y 599.939,Z 685.03,A -85,B 0,C 180,E1 1081.438,E2 1081.438} C_VEL
LIN {X 0,Y 599.965,Z 685.03,A -85,B 0,C 180,E1 1085.771,E2 1085.771} C_VEL
LIN {X 0,Y 599.628,Z 685.03,A -85,B 0,C 180,E1 1091.611,E2 1091.611} C_VEL
LIN {X 0,Y 599.7,Z 685.03,A -85,B 0,C 180,E1 1096.064,E2 1096.064} C_VEL
LIN {X 0,Y 599.531,Z 685.03,A -85,B 0,C 180,E1 1101.366,E2 1101.366} C_VEL
LIN {X 0,Y 599.775,Z 685.03,A -85,B 0,C 180,E1 1105.317,E2 1105.317} C_VEL
LIN {X 0,Y 599.491,Z 685.03,A -85,B 0,C 180,E1 1111.149,E2 1111.149} C_VEL
LIN {X 0,Y 599.655,Z 685.03,A -85,B 0,C 180,E1 1117.146,E2 1117.146} C_VEL
LIN {X 0,Y 599.542,Z 685.03,A -85,B 0,C 180,E1 1123.122,E2 1123.122} C_VEL
LIN {X 0,Y 599.394,Z 685.03,A -85,B 0,C 180,E1 1129.114,E2 1129.114} C_VEL
LIN {X 0,Y 599.295,Z 685.03,A -85,B 0,C 180,E1 1133.672,E2 1133.672} C_VEL
LIN {X 0,Y 599.64,Z 685.03,A -85,B 0,C 180,E1 1138.098,E2 1138.098} C_VEL
LIN {X 0,Y 599.557,Z 685.03,A -85,B 0,C 180,E1 1143.062,E2 1143.062} C_VEL
LIN {X 0,Y 599.844,Z 685.579,A -85,B 0,C 180,E1 1145.895,E2 1145.895} C_VEL
LIN {X 0,Y 601.088,Z 700.867,A -85,B 0,C 180,E1 1146.543,E2 1146.543} C_VEL
LIN {X 0,Y 600.751,Z 736.528,A -85,B 0,C 180,E1 1148.403,E2 1148.403} C_VEL
LIN {X 0,Y 600.491,Z 767.887,A -85,B 0,C 180,E1 1150.684,E2 1150.684} C_VEL
LIN {X 0,Y 600.217,Z 796.757,A -85,B 0,C 180,E1 1153.509,E2 1153.509} C_VEL
LIN {X 0,Y 600.041,Z 819.799,A -85,B 0,C 180,E1 1156.549,E2 1156.549} C_VEL
LIN {X 0,Y 599.95,Z 838.1,A -85,B 0,C 180,E1 1159.859,E2 1159.859} C_VEL
LIN {X 0,Y 599.931,Z 851.043,A -85,B 0,C 180,E1 1163.324,E2 1163.324} C_VEL
LIN {X 0,Y 600.002,Z 858.731,A -85,B 0,C 180,E1 1167.117,E2 1167.117} C_VEL
LIN {X 0,Y 599.851,Z 860.496,A -85,B 0,C 180,E1 1170,E2 1170} C_VEL
LIN {X 0,Y 599.944,Z 857.612,A -85,B 0,C 180,E1 1173.605,E2 1173.605} C_VEL
LIN {X 0,Y 599.927,Z 849.04,A -85,B 0,C 180,E1 1177.225,E2 1177.225} C_VEL
LIN {X 0,Y 600.036,Z 834.929,A -85,B 0,C 180,E1 1180.716,E2 1180.716} C_VEL
LIN {X 0,Y 600.125,Z 815.5,A -85,B 0,C 180,E1 1184.006,E2 1184.006} C_VEL
LIN {X 0,Y 600.282,Z 791.794,A -85,B 0,C 180,E1 1186.946,E2 1186.946} C_VEL
LIN {X 0,Y 600.545,Z 762.805,A -85,B 0,C 180,E1 1189.649,E2 1189.649} C_VEL
LIN {X 0,Y 600.786,Z 730.128,A -85,B 0,C 180,E1 1191.893,E2 1191.893} C_VEL
LIN {X 0,Y 600.878,Z 695.524,A -85,B 0,C 180,E1 1193.593,E2 1193.593} C_VEL
LIN {X 0,Y 599.832,Z 685.03,A -85,B 0,C 180,E1 1194.069,E2 1194.069} C_VEL
LIN {X 0,Y 599.664,Z 685.03,A -85,B 0,C 180,E1 1198.562,E2 1198.562} C_VEL
LIN {X 0,Y 599.685,Z 685.03,A -85,B 0,C 180,E1 1203.873,E2 1203.873} C_VEL
LIN {X 0,Y 599.629,Z 685.03,A -85,B 0,C 180,E1 1208.986,E2 1208.986} C_VEL
LIN {X 0,Y 599.511,Z 685.03,A -85,B 0,C 180,E1 1215.197,E2 1215.197} C_VEL
LIN {X 0,Y 599.513,Z 685.03,A -85,B 0,C 180,E1 1221.012,E2 1221.012} C_VEL
LIN {X 0,Y 599.554,Z 685.03,A -85,B 0,C 180,E1 1224.635,E2 1224.635} C_VEL
LIN {X 0,Y 599.589,Z 685.03,A -85,B 0,C 180,E1 1229.784,E2 1229.784} C_VEL
LIN {X 0,Y 599.852,Z 685.03,A -85,B 0,C 180,E1 1234.907,E2 1234.907} C_VEL
LIN {X 0,Y 599.72,Z 685.03,A -85,B 0,C 180,E1 1240.911,E2 1240.911} C_VEL
LIN {X 0,Y 599.966,Z 685.03,A -85,B 0,C 180,E1 1246.921,E2 1246.921} C_VEL
LIN {X 0,Y 599.676,Z 685.03,A -85,B 0,C 180,E1 1252.775,E2 1252.775} C_VEL
LIN {X 0,Y 599.8,Z 685.03,A -85,B 0,C 180,E1 1257.119,E2 1257.119} C_VEL
LIN {X 0,Y 599.56,Z 685.03,A -85,B 0,C 180,E1 1259.16,E2 1259.16} C_VEL
LIN {X 0,Y 597.184,Z 685.03,A -85,B 0,C 180,E1 1260.396,E2 1260.396} C_VEL
LIN {X 0,Y 591.771,Z 685.03,A -85,B 0,C 180,E1 1262.458,E2 1262.458} C_VEL
LIN {X 0,Y 591.665,Z 685.03,A -85,B 0,C 180,E1 1267.329,E2 1267.329} C_VEL
LIN {X 0,Y 591.66,Z 685.03,A -85,B 0,C 180,E1 1271.775,E2 1271.775} C_VEL
LIN {X 0,Y 591.717,Z 685.03,A -85,B 0,C 180,E1 1276.293,E2 1276.293} C_VEL
LIN {X 0,Y 591.745,Z 685.03,A -85,B 0,C 180,E1 1280.918,E2 1280.918} C_VEL
LIN {X 0,Y 591.57,Z 685.03,A -85,B 0,C 180,E1 1286.774,E2 1286.774} C_VEL
LIN {X 0,Y 591.596,Z 685.03,A -85,B 0,C 180,E1 1290.674,E2 1290.674} C_VEL
LIN {X 0,Y 591.659,Z 685.03,A -85,B 0,C 180,E1 1295.917,E2 1295.917} C_VEL
LIN {X 0,Y 591.564,Z 685.03,A -85,B 0,C 180,E1 1302.29,E2 1302.29} C_VEL
LIN {X 0,Y 591.605,Z 685.03,A -85,B 0,C 180,E1 1308.458,E2 1308.458} C_VEL
LIN {X 0,Y 591.787,Z 685.03,A -85,B 0,C 180,E1 1314.093,E2 1314.093} C_VEL
LIN {X 0,Y 591.986,Z 685.299,A -85,B 0,C 180,E1 1319.298,E2 1319.298} C_VEL
LIN {X 0,Y 594.687,Z 694.975,A -85,B 0,C 180,E1 1319.585,E2 1319.585} C_VEL
LIN {X 0,Y 594.681,Z 773.257,A -85,B 0,C 180,E1 1320.762,E2 1320.762} C_VEL
LIN {X 0,Y 594.436,Z 810.286,A -85,B 0,C 180,E1 1321.859,E2 1321.859} C_VEL
LIN {X 0,Y 594.009,Z 844.942,A -85,B 0,C 180,E1 1323.401,E2 1323.401} C_VEL
LIN {X 0,Y 593.457,Z 879.782,A -85,B 0,C 180,E1 1325.536,E2 1325.536} C_VEL
LIN {X 0,Y 592.98,Z 911.333,A -85,B 0,C 180,E1 1328.095,E2 1328.095} C_VEL
LIN {X 0,Y 592.557,Z 939.519,A -85,B 0,C 180,E1 1331.053,E2 1331.053} C_VEL
LIN {X 0,Y 592.16,Z 963.335,A -85,B 0,C 180,E1 1334.291,E2 1334.291} C_VEL
LIN {X 0,Y 592.042,Z 981.278,A -85,B 0,C 180,E1 1337.488,E2 1337.488} C_VEL
LIN {X 0,Y 592.047,Z 995.073,A -85,B 0,C 180,E1 1340.834,E2 1340.834} C_VEL
LIN {X 0,Y 592.037,Z 1004.22,A -85,B 0,C 180,E1 1344.148,E2 1344.148} C_VEL
LIN {X 0,Y 592.065,Z 1008.906,A -85,B 0,C 180,E1 1347.078,E2 1347.078} C_VEL
LIN {X 0,Y 591.932,Z 1010.5,A -85,B 0,C 180,E1 1350,E2 1350} C_VEL
LIN {X 0,Y 591.893,Z 1008.906,A -85,B 0,C 180,E1 1352.923,E2 1352.923} C_VEL
LIN {X 0,Y 591.951,Z 1002.581,A -85,B 0,C 180,E1 1356.593,E2 1356.593} C_VEL
LIN {X 0,Y 591.956,Z 991.046,A -85,B 0,C 180,E1 1360.279,E2 1360.279} C_VEL
LIN {X 0,Y 592.143,Z 974.319,A -85,B 0,C 180,E1 1363.867,E2 1363.867} C_VEL
LIN {X 0,Y 592.378,Z 952.739,A -85,B 0,C 180,E1 1367.265,E2 1367.265} C_VEL
LIN {X 0,Y 592.782,Z 925.46,A -85,B 0,C 180,E1 1370.521,E2 1370.521} C_VEL
LIN {X 0,Y 593.256,Z 893.696,A -85,B 0,C 180,E1 1373.416,E2 1373.416} C_VEL
LIN {X 0,Y 593.745,Z 859.244,A -85,B 0,C 180,E1 1375.8,E2 1375.8} C_VEL
LIN {X 0,Y 594.251,Z 822.523,A -85,B 0,C 180,E1 1377.659,E2 1377.659} C_VEL
LIN {X 0,Y 594.591,Z 784.327,A -85,B 0,C 180,E1 1378.967,E2 1378.967} C_VEL
LIN {X 0,Y 594.89,Z 744.094,A -85,B 0,C 180,E1 1379.732,E2 1379.732} C_VEL
LIN {X 0,Y 594.005,Z 691.202,A -85,B 0,C 180,E1 1380.505,E2 1380.505} C_VEL
LIN {X 0,Y 591.966,Z 685.03,A -85,B 0,C 180,E1 1380.771,E2 1380.771} C_VEL
LIN {X 0,Y 591.761,Z 685.03,A -85,B 0,C 180,E1 1385.909,E2 1385.909} C_VEL
LIN {X 0,Y 591.59,Z 685.03,A -85,B 0,C 180,E1 1392.293,E2 1392.293} C_VEL
LIN {X 0,Y 591.632,Z 685.03,A -85,B 0,C 180,E1 1398.46,E2 1398.46} C_VEL
LIN {X 0,Y 591.737,Z 685.03,A -85,B 0,C 180,E1 1404.089,E2 1404.089} C_VEL
LIN {X 0,Y 591.592,Z 685.03,A -85,B 0,C 180,E1 1409.326,E2 1409.326} C_VEL
LIN {X 0,Y 591.469,Z 685.03,A -85,B 0,C 180,E1 1414.295,E2 1414.295} C_VEL
LIN {X 0,Y 591.493,Z 685.03,A -85,B 0,C 180,E1 1419.073,E2 1419.073} C_VEL
LIN {X 0,Y 591.685,Z 685.03,A -85,B 0,C 180,E1 1423.706,E2 1423.706} C_VEL
LIN {X 0,Y 591.694,Z 685.03,A -85,B 0,C 180,E1 1428.226,E2 1428.226} C_VEL
LIN {X 0,Y 591.767,Z 685.03,A -85,B 0,C 180,E1 1432.673,E2 1432.673} C_VEL
LIN {X 0,Y 591.926,Z 685.03,A -85,B 0,C 180,E1 1437.075,E2 1437.075} C_VEL
LIN {X 0,Y 592.029,Z 685.03,A -85,B 0,C 180,E1 1441.458,E2 1441.458} C_VEL
LIN {X 0,Y 591.93,Z 685.03,A -85,B 0,C 180,E1 1446.165,E2 1446.165} C_VEL
LIN {X 0,Y 591.694,Z 685.03,A -85,B 0,C 180,E1 1451.769,E2 1451.769} C_VEL
LIN {X 0,Y 591.755,Z 685.03,A -85,B 0,C 180,E1 1456.286,E2 1456.286} C_VEL
LIN {X 0,Y 591.758,Z 685.03,A -85,B 0,C 180,E1 1460.912,E2 1460.912} C_VEL
LIN {X 0,Y 591.549,Z 685.03,A -85,B 0,C 180,E1 1466.77,E2 1466.77} C_VEL
LIN {X 0,Y 591.618,Z 685.03,A -85,B 0,C 180,E1 1470.666,E2 1470.666} C_VEL
LIN {X 0,Y 591.703,Z 685.03,A -85,B 0,C 180,E1 1475.907,E2 1475.907} C_VEL
LIN {X 0,Y 591.61,Z 685.03,A -85,B 0,C 180,E1 1481.535,E2 1481.535} C_VEL
LIN {X 0,Y 591.481,Z 685.03,A -85,B 0,C 180,E1 1486.463,E2 1486.463} C_VEL
LIN {X 0,Y 591.511,Z 685.03,A -85,B 0,C 180,E1 1492.254,E2 1492.254} C_VEL
LIN {X 0,Y 591.72,Z 685.03,A -85,B 0,C 180,E1 1497.62,E2 1497.62} C_VEL
LIN {X 0,Y 591.66,Z 685.03,A -85,B 0,C 180,E1 1503.194,E2 1503.194} C_VEL
LIN {X 0,Y 591.86,Z 685.03,A -85,B 0,C 180,E1 1505.527,E2 1505.527} C_VEL
LIN {X 0,Y 593.774,Z 697.539,A -85,B 0,C 180,E1 1506.1,E2 1506.1} C_VEL
LIN {X 0,Y 593.365,Z 733.296,A -85,B 0,C 180,E1 1507.914,E2 1507.914} C_VEL
LIN {X 0,Y 592.93,Z 765.632,A -85,B 0,C 180,E1 1510.237,E2 1510.237} C_VEL
LIN {X 0,Y 592.51,Z 793.824,A -85,B 0,C 180,E1 1512.955,E2 1512.955} C_VEL
LIN {X 0,Y 592.24,Z 818.11,A -85,B 0,C 180,E1 1516.106,E2 1516.106} C_VEL
LIN {X 0,Y 592.058,Z 835.848,A -85,B 0,C 180,E1 1519.243,E2 1519.243} C_VEL
LIN {X 0,Y 591.995,Z 849.322,A -85,B 0,C 180,E1 1522.678,E2 1522.678} C_VEL
LIN {X 0,Y 592.042,Z 857.761,A -85,B 0,C 180,E1 1526.347,E2 1526.347} C_VEL
LIN {X 0,Y 591.952,Z 860.496,A -85,B 0,C 180,E1 1530,E2 1530} C_VEL
LIN {X 0,Y 592.055,Z 857.614,A -85,B 0,C 180,E1 1533.653,E2 1533.653} C_VEL
LIN {X 0,Y 592.055,Z 849.043,A -85,B 0,C 180,E1 1537.321,E2 1537.321} C_VEL
LIN {X 0,Y 592.168,Z 835.289,A -85,B 0,C 180,E1 1540.784,E2 1540.784} C_VEL
LIN {X 0,Y 592.316,Z 815.21,A -85,B 0,C 180,E1 1544.236,E2 1544.236} C_VEL
LIN {X 0,Y 592.616,Z 790.378,A -85,B 0,C 180,E1 1547.328,E2 1547.328} C_VEL
LIN {X 0,Y 592.984,Z 761.411,A -85,B 0,C 180,E1 1550.023,E2 1550.023} C_VEL
LIN {X 0,Y 593.366,Z 729.913,A -85,B 0,C 180,E1 1552.194,E2 1552.194} C_VEL
LIN {X 0,Y 593.533,Z 694.476,A -85,B 0,C 180,E1 1553.947,E2 1553.947} C_VEL
LIN {X 0,Y 591.907,Z 685.03,A -85,B 0,C 180,E1 1554.395,E2 1554.395} C_VEL
LIN {X 0,Y 591.5,Z 685.03,A -85,B 0,C 180,E1 1559.857,E2 1559.857} C_VEL
LIN {X 0,Y 591.733,Z 685.03,A -85,B 0,C 180,E1 1564.127,E2 1564.127} C_VEL
LIN {X 0,Y 591.523,Z 685.03,A -85,B 0,C 180,E1 1570.075,E2 1570.075} C_VEL
LIN {X 0,Y 591.575,Z 685.03,A -85,B 0,C 180,E1 1575.58,E2 1575.58} C_VEL
LIN {X 0,Y 591.561,Z 685.03,A -85,B 0,C 180,E1 1580.385,E2 1580.385} C_VEL
LIN {X 0,Y 591.637,Z 685.03,A -85,B 0,C 180,E1 1584.703,E2 1584.703} C_VEL
LIN {X 0,Y 591.543,Z 685.03,A -85,B 0,C 180,E1 1591.014,E2 1591.014} C_VEL
LIN {X 0,Y 591.65,Z 685.03,A -85,B 0,C 180,E1 1595.921,E2 1595.921} C_VEL
LIN {X 0,Y 591.822,Z 685.03,A -85,B 0,C 180,E1 1600.647,E2 1600.647} C_VEL
LIN {X 0,Y 592.02,Z 685.03,A -85,B 0,C 180,E1 1606.742,E2 1606.742} C_VEL
LIN {X 0,Y 591.788,Z 685.03,A -85,B 0,C 180,E1 1612.716,E2 1612.716} C_VEL
LIN {X 0,Y 591.893,Z 685.03,A -85,B 0,C 180,E1 1617.08,E2 1617.08} C_VEL
LIN {X 0,Y 591.771,Z 685.03,A -85,B 0,C 180,E1 1622.458,E2 1622.458} C_VEL
LIN {X 0,Y 587.718,Z 685.03,A -85,B 0,C 180,E1 1624.115,E2 1624.115} C_VEL
LIN {X 0,Y 584.063,Z 685.03,A -85,B 0,C 180,E1 1625.793,E2 1625.793} C_VEL
LIN {X 0,Y 583.754,Z 685.03,A -85,B 0,C 180,E1 1631.937,E2 1631.937} C_VEL
LIN {X 0,Y 583.702,Z 685.03,A -85,B 0,C 180,E1 1636.956,E2 1636.956} C_VEL
LIN {X 0,Y 583.706,Z 685.03,A -85,B 0,C 180,E1 1641.461,E2 1641.461} C_VEL
LIN {X 0,Y 583.781,Z 685.03,A -85,B 0,C 180,E1 1646.068,E2 1646.068} C_VEL
LIN {X 0,Y 583.547,Z 685.03,A -85,B 0,C 180,E1 1651.423,E2 1651.423} C_VEL
LIN {X 0,Y 583.618,Z 685.03,A -85,B 0,C 180,E1 1656.724,E2 1656.724} C_VEL
LIN {X 0,Y 583.659,Z 685.03,A -85,B 0,C 180,E1 1662.237,E2 1662.237} C_VEL
LIN {X 0,Y 583.69,Z 685.03,A -85,B 0,C 180,E1 1668.566,E2 1668.566} C_VEL
LIN {X 0,Y 583.8,Z 685.03,A -85,B 0,C 180,E1 1673.523,E2 1673.523} C_VEL
LIN {X 0,Y 584.021,Z 685.032,A -85,B 0,C 180,E1 1678.829,E2 1678.829} C_VEL
LIN {X 0,Y 587.87,Z 697.24,A -85,B 0,C 180,E1 1679.226,E2 1679.226} C_VEL
LIN {X 0,Y 587.773,Z 773.36,A -85,B 0,C 180,E1 1680.387,E2 1680.387} C_VEL
LIN {X 0,Y 587.384,Z 810.634,A -85,B 0,C 180,E1 1681.504,E2 1681.504} C_VEL
LIN {X 0,Y 586.783,Z 847.105,A -85,B 0,C 180,E1 1683.167,E2 1683.167} C_VEL
LIN {X 0,Y 586.024,Z 882.423,A -85,B 0,C 180,E1 1685.401,E2 1685.401} C_VEL
LIN {X 0,Y 585.363,Z 914.817,A -85,B 0,C 180,E1 1688.128,E2 1688.128} C_VEL
LIN {X 0,Y 584.789,Z 944.306,A -85,B 0,C 180,E1 1691.378,E2 1691.378} C_VEL
LIN {X 0,Y 584.391,Z 968.075,A -85,B 0,C 180,E1 1694.844,E2 1694.844} C_VEL
LIN {X 0,Y 584.146,Z 987.045,A -85,B 0,C 180,E1 1698.599,E2 1698.599} C_VEL
LIN {X 0,Y 584.101,Z 999.718,A -85,B 0,C 180,E1 1702.205,E2 1702.205} C_VEL
LIN {X 0,Y 583.996,Z 1006.956,A -85,B 0,C 180,E1 1705.554,E2 1705.554} C_VEL
LIN {X 0,Y 584.027,Z 1010.086,A -85,B 0,C 180,E1 1708.519,E2 1708.519} C_VEL
LIN {X 0,Y 584.185,Z 1010.086,A -85,B 0,C 180,E1 1711.48,E2 1711.48} C_VEL
LIN {X 0,Y 584.209,Z 1005.757,A -85,B 0,C 180,E1 1715.187,E2 1715.187} C_VEL
LIN {X 0,Y 584.197,Z 995.073,A -85,B 0,C 180,E1 1719.29,E2 1719.29} C_VEL
LIN {X 0,Y 584.316,Z 979.45,A -85,B 0,C 180,E1 1723.06,E2 1723.06} C_VEL
LIN {X 0,Y 584.557,Z 958.38,A -85,B 0,C 180,E1 1726.686,E2 1726.686} C_VEL
LIN {X 0,Y 585.024,Z 932.787,A -85,B 0,C 180,E1 1729.994,E2 1729.994} C_VEL
LIN {X 0,Y 585.594,Z 903.859,A -85,B 0,C 180,E1 1732.878,E2 1732.878} C_VEL
LIN {X 0,Y 586.296,Z 870.586,A -85,B 0,C 180,E1 1735.424,E2 1735.424} C_VEL
LIN {X 0,Y 586.972,Z 836.095,A -85,B 0,C 180,E1 1737.4,E2 1737.4} C_VEL
LIN {X 0,Y 587.53,Z 798.85,A -85,B 0,C 180,E1 1738.911,E2 1738.911} C_VEL
LIN {X 0,Y 587.995,Z 762.807,A -85,B 0,C 180,E1 1739.826,E2 1739.826} C_VEL
LIN {X 0,Y 587.268,Z 693.533,A -85,B 0,C 180,E1 1740.861,E2 1740.861} C_VEL
LIN {X 0,Y 584.071,Z 685.03,A -85,B 0,C 180,E1 1741.21,E2 1741.21} C_VEL
LIN {X 0,Y 583.801,Z 685.03,A -85,B 0,C 180,E1 1746.748,E2 1746.748} C_VEL
LIN {X 0,Y 583.689,Z 685.03,A -85,B 0,C 180,E1 1752.235,E2 1752.235} C_VEL
LIN {X 0,Y 583.715,Z 685.03,A -85,B 0,C 180,E1 1758.564,E2 1758.564} C_VEL
LIN {X 0,Y 583.76,Z 685.03,A -85,B 0,C 180,E1 1763.52,E2 1763.52} C_VEL
LIN {X 0,Y 583.68,Z 685.03,A -85,B 0,C 180,E1 1768.556,E2 1768.556} C_VEL
LIN {X 0,Y 583.552,Z 685.03,A -85,B 0,C 180,E1 1773.921,E2 1773.921} C_VEL
LIN {X 0,Y 583.579,Z 685.03,A -85,B 0,C 180,E1 1778.775,E2 1778.775} C_VEL
LIN {X 0,Y 583.784,Z 685.03,A -85,B 0,C 180,E1 1783.479,E2 1783.479} C_VEL
LIN {X 0,Y 583.812,Z 685.03,A -85,B 0,C 180,E1 1788.064,E2 1788.064} C_VEL
LIN {X 0,Y 583.858,Z 685.03,A -85,B 0,C 180,E1 1792.573,E2 1792.573} C_VEL
LIN {X 0,Y 584.04,Z 685.03,A -85,B 0,C 180,E1 1797.035,E2 1797.035} C_VEL
LIN {X 0,Y 584.138,Z 685.03,A -85,B 0,C 180,E1 1801.477,E2 1801.477} C_VEL
LIN {X 0,Y 584.114,Z 685.03,A -85,B 0,C 180,E1 1805.928,E2 1805.928} C_VEL
LIN {X 0,Y 583.782,Z 685.03,A -85,B 0,C 180,E1 1811.93,E2 1811.93} C_VEL
LIN {X 0,Y 583.719,Z 685.03,A -85,B 0,C 180,E1 1816.962,E2 1816.962} C_VEL
LIN {X 0,Y 583.718,Z 685.03,A -85,B 0,C 180,E1 1821.464,E2 1821.464} C_VEL
LIN {X 0,Y 583.774,Z 685.03,A -85,B 0,C 180,E1 1826.062,E2 1826.062} C_VEL
LIN {X 0,Y 583.561,Z 685.03,A -85,B 0,C 180,E1 1831.425,E2 1831.425} C_VEL
LIN {X 0,Y 583.736,Z 685.03,A -85,B 0,C 180,E1 1836.739,E2 1836.739} C_VEL
LIN {X 0,Y 583.709,Z 685.03,A -85,B 0,C 180,E1 1842.225,E2 1842.225} C_VEL
LIN {X 0,Y 583.52,Z 685.03,A -85,B 0,C 180,E1 1847.75,E2 1847.75} C_VEL
LIN {X 0,Y 583.502,Z 685.03,A -85,B 0,C 180,E1 1853.281,E2 1853.281} C_VEL
LIN {X 0,Y 583.852,Z 685.03,A -85,B 0,C 180,E1 1857.129,E2 1857.129} C_VEL
LIN {X 0,Y 583.748,Z 685.03,A -85,B 0,C 180,E1 1862.27,E2 1862.27} C_VEL
LIN {X 0,Y 583.87,Z 685.03,A -85,B 0,C 180,E1 1865.17,E2 1865.17} C_VEL
LIN {X 0,Y 586.461,Z 698.467,A -85,B 0,C 180,E1 1865.822,E2 1865.822} C_VEL
LIN {X 0,Y 585.907,Z 733.904,A -85,B 0,C 180,E1 1867.658,E2 1867.658} C_VEL
LIN {X 0,Y 585.349,Z 765.445,A -85,B 0,C 180,E1 1869.954,E2 1869.954} C_VEL
LIN {X 0,Y 584.762,Z 793.462,A -85,B 0,C 180,E1 1872.683,E2 1872.683} C_VEL
LIN {X 0,Y 584.459,Z 816.744,A -85,B 0,C 180,E1 1875.702,E2 1875.702} C_VEL
LIN {X 0,Y 584.238,Z 835.022,A -85,B 0,C 180,E1 1878.919,E2 1878.919} C_VEL
LIN {X 0,Y 584.144,Z 848.177,A -85,B 0,C 180,E1 1882.206,E2 1882.206} C_VEL
LIN {X 0,Y 584.099,Z 856.566,A -85,B 0,C 180,E1 1885.555,E2 1885.555} C_VEL
LIN {X 0,Y 584.068,Z 860.042,A -85,B 0,C 180,E1 1888.52,E2 1888.52} C_VEL
LIN {X 0,Y 584.154,Z 859.981,A -85,B 0,C 180,E1 1891.48,E2 1891.48} C_VEL
LIN {X 0,Y 584.157,Z 854.895,A -85,B 0,C 180,E1 1895.187,E2 1895.187} C_VEL
LIN {X 0,Y 584.189,Z 843.946,A -85,B 0,C 180,E1 1898.916,E2 1898.916} C_VEL
LIN {X 0,Y 584.321,Z 828.282,A -85,B 0,C 180,E1 1902.301,E2 1902.301} C_VEL
LIN {X 0,Y 584.611,Z 807.3,A -85,B 0,C 180,E1 1905.533,E2 1905.533} C_VEL
LIN {X 0,Y 585.051,Z 782.185,A -85,B 0,C 180,E1 1908.419,E2 1908.419} C_VEL
LIN {X 0,Y 585.594,Z 751.655,A -85,B 0,C 180,E1 1911.048,E2 1911.048} C_VEL
LIN {X 0,Y 586.139,Z 718.175,A -85,B 0,C 180,E1 1913.15,E2 1913.15} C_VEL
LIN {X 0,Y 585.776,Z 691.928,A -85,B 0,C 180,E1 1914.392,E2 1914.392} C_VEL
LIN {X 0,Y 583.955,Z 685.03,A -85,B 0,C 180,E1 1914.784,E2 1914.784} C_VEL
LIN {X 0,Y 583.654,Z 685.03,A -85,B 0,C 180,E1 1919.421,E2 1919.421} C_VEL
LIN {X 0,Y 583.725,Z 685.03,A -85,B 0,C 180,E1 1924.661,E2 1924.661} C_VEL
LIN {X 0,Y 583.589,Z 685.03,A -85,B 0,C 180,E1 1930.273,E2 1930.273} C_VEL
LIN {X 0,Y 583.704,Z 685.03,A -85,B 0,C 180,E1 1936.374,E2 1936.374} C_VEL
LIN {X 0,Y 583.688,Z 685.03,A -85,B 0,C 180,E1 1941.657,E2 1941.657} C_VEL
LIN {X 0,Y 583.499,Z 685.03,A -85,B 0,C 180,E1 1947.112,E2 1947.112} C_VEL
LIN {X 0,Y 583.601,Z 685.03,A -85,B 0,C 180,E1 1952.268,E2 1952.268} C_VEL
LIN {X 0,Y 583.604,Z 685.03,A -85,B 0,C 180,E1 1957.184,E2 1957.184} C_VEL
LIN {X 0,Y 583.832,Z 685.03,A -85,B 0,C 180,E1 1961.936,E2 1961.936} C_VEL
LIN {X 0,Y 584.101,Z 685.03,A -85,B 0,C 180,E1 1966.559,E2 1966.559} C_VEL
LIN {X 0,Y 583.864,Z 685.03,A -85,B 0,C 180,E1 1972.7,E2 1972.7} C_VEL
LIN {X 0,Y 584.01,Z 685.03,A -85,B 0,C 180,E1 1977.041,E2 1977.041} C_VEL
LIN {X 0,Y 583.889,Z 685.03,A -85,B 0,C 180,E1 1982.443,E2 1982.443} C_VEL
LIN {X 0,Y 584.063,Z 685.03,A -85,B 0,C 180,E1 1985.793,E2 1985.793} C_VEL
LIN {X 0,Y 581.601,Z 685.03,A -85,B 0,C 180,E1 1987.054,E2 1987.054} C_VEL
LIN {X 0,Y 575.942,Z 685.03,A -85,B 0,C 180,E1 1988.939,E2 1988.939} C_VEL
LIN {X 0,Y 575.839,Z 685.03,A -85,B 0,C 180,E1 1989.158,E2 1989.158} C_VEL
LIN {X 0,Y 575.92,Z 685.03,A -85,B 0,C 180,E1 1995.191,E2 1995.191} C_VEL
LIN {X 0,Y 575.79,Z 685.03,A -85,B 0,C 180,E1 2001.526,E2 2001.526} C_VEL
LIN {X 0,Y 575.71,Z 685.03,A -85,B 0,C 180,E1 2006.979,E2 2006.979} C_VEL
LIN {X 0,Y 575.639,Z 685.03,A -85,B 0,C 180,E1 2011.621,E2 2011.621} C_VEL
LIN {X 0,Y 575.658,Z 685.03,A -85,B 0,C 180,E1 2017.079,E2 2017.079} C_VEL
LIN {X 0,Y 575.675,Z 685.03,A -85,B 0,C 180,E1 2022.963,E2 2022.963} C_VEL
LIN {X 0,Y 575.747,Z 685.03,A -85,B 0,C 180,E1 2029.063,E2 2029.063} C_VEL
LIN {X 0,Y 575.931,Z 685.03,A -85,B 0,C 180,E1 2034.801,E2 2034.801} C_VEL
LIN {X 0,Y 576.085,Z 685.051,A -85,B 0,C 180,E1 2038.351,E2 2038.351} C_VEL
LIN {X 0,Y 581.087,Z 699.31,A -85,B 0,C 180,E1 2038.856,E2 2038.856} C_VEL
LIN {X 0,Y 580.916,Z 773.324,A -85,B 0,C 180,E1 2040.001,E2 2040.001} C_VEL
LIN {X 0,Y 580.389,Z 810.984,A -85,B 0,C 180,E1 2041.141,E2 2041.141} C_VEL
LIN {X 0,Y 579.574,Z 846.92,A -85,B 0,C 180,E1 2042.795,E2 2042.795} C_VEL
LIN {X 0,Y 578.67,Z 881.902,A -85,B 0,C 180,E1 2045.027,E2 2045.027} C_VEL
LIN {X 0,Y 577.84,Z 913.674,A -85,B 0,C 180,E1 2047.717,E2 2047.717} C_VEL
LIN {X 0,Y 577.094,Z 943.095,A -85,B 0,C 180,E1 2050.968,E2 2050.968} C_VEL
LIN {X 0,Y 576.553,Z 968.076,A -85,B 0,C 180,E1 2054.633,E2 2054.633} C_VEL
LIN {X 0,Y 576.273,Z 986.767,A -85,B 0,C 180,E1 2058.372,E2 2058.372} C_VEL
LIN {X 0,Y 576.206,Z 999.718,A -85,B 0,C 180,E1 2062.097,E2 2062.097} C_VEL
LIN {X 0,Y 576.097,Z 1006.956,A -85,B 0,C 180,E1 2065.493,E2 2065.493} C_VEL
LIN {X 0,Y 576.127,Z 1010.086,A -85,B 0,C 180,E1 2068.499,E2 2068.499} C_VEL
LIN {X 0,Y 576.279,Z 1010.087,A -85,B 0,C 180,E1 2071.5,E2 2071.5} C_VEL
LIN {X 0,Y 576.251,Z 1004.868,A -85,B 0,C 180,E1 2075.698,E2 2075.698} C_VEL
LIN {X 0,Y 576.289,Z 995.073,A -85,B 0,C 180,E1 2079.419,E2 2079.419} C_VEL
LIN {X 0,Y 576.454,Z 979.449,A -85,B 0,C 180,E1 2083.241,E2 2083.241} C_VEL
LIN {X 0,Y 576.774,Z 958.378,A -85,B 0,C 180,E1 2086.918,E2 2086.918} C_VEL
LIN {X 0,Y 577.379,Z 932.871,A -85,B 0,C 180,E1 2090.261,E2 2090.261} C_VEL
LIN {X 0,Y 578.124,Z 902.631,A -85,B 0,C 180,E1 2093.301,E2 2093.301} C_VEL
LIN {X 0,Y 579.049,Z 868.677,A -85,B 0,C 180,E1 2095.896,E2 2095.896} C_VEL
LIN {X 0,Y 579.918,Z 832.761,A -85,B 0,C 180,E1 2097.929,E2 2097.929} C_VEL
LIN {X 0,Y 580.592,Z 794.736,A -85,B 0,C 180,E1 2099.425,E2 2099.425} C_VEL
LIN {X 0,Y 581.194,Z 757.162,A -85,B 0,C 180,E1 2100.305,E2 2100.305} C_VEL
LIN {X 0,Y 580.604,Z 696.37,A -85,B 0,C 180,E1 2101.214,E2 2101.214} C_VEL
LIN {X 0,Y 576.131,Z 685.03,A -85,B 0,C 180,E1 2101.689,E2 2101.689} C_VEL
LIN {X 0,Y 575.878,Z 685.03,A -85,B 0,C 180,E1 2107.062,E2 2107.062} C_VEL
LIN {X 0,Y 575.683,Z 685.03,A -85,B 0,C 180,E1 2112.962,E2 2112.962} C_VEL
LIN {X 0,Y 575.762,Z 685.03,A -85,B 0,C 180,E1 2119.064,E2 2119.064} C_VEL
LIN {X 0,Y 575.878,Z 685.03,A -85,B 0,C 180,E1 2124.797,E2 2124.797} C_VEL
LIN {X 0,Y 575.751,Z 685.03,A -85,B 0,C 180,E1 2130.133,E2 2130.133} C_VEL
LIN {X 0,Y 575.69,Z 685.03,A -85,B 0,C 180,E1 2135.203,E2 2135.203} C_VEL
LIN {X 0,Y 575.932,Z 685.03,A -85,B 0,C 180,E1 2141.673,E2 2141.673} C_VEL
LIN {X 0,Y 575.908,Z 685.03,A -85,B 0,C 180,E1 2147.898,E2 2147.898} C_VEL
LIN {X 0,Y 575.954,Z 685.03,A -85,B 0,C 180,E1 2152.47,E2 2152.47} C_VEL
LIN {X 0,Y 576.13,Z 685.03,A -85,B 0,C 180,E1 2156.995,E2 2156.995} C_VEL
LIN {X 0,Y 576.228,Z 685.03,A -85,B 0,C 180,E1 2161.498,E2 2161.498} C_VEL
LIN {X 0,Y 576.209,Z 685.03,A -85,B 0,C 180,E1 2166.01,E2 2166.01} C_VEL
LIN {X 0,Y 575.856,Z 685.03,A -85,B 0,C 180,E1 2172.097,E2 2172.097} C_VEL
LIN {X 0,Y 575.879,Z 685.03,A -85,B 0,C 180,E1 2176.748,E2 2176.748} C_VEL
LIN {X 0,Y 575.825,Z 685.03,A -85,B 0,C 180,E1 2181.519,E2 2181.519} C_VEL
LIN {X 0,Y 575.69,Z 685.03,A -85,B 0,C 180,E1 2186.975,E2 2186.975} C_VEL
LIN {X 0,Y 575.653,Z 685.03,A -85,B 0,C 180,E1 2191.613,E2 2191.613} C_VEL
LIN {X 0,Y 575.816,Z 685.03,A -85,B 0,C 180,E1 2197.06,E2 2197.06} C_VEL
LIN {X 0,Y 575.771,Z 685.03,A -85,B 0,C 180,E1 2202.946,E2 2202.946} C_VEL
LIN {X 0,Y 575.627,Z 685.03,A -85,B 0,C 180,E1 2209.052,E2 2209.052} C_VEL
LIN {X 0,Y 575.697,Z 685.03,A -85,B 0,C 180,E1 2214.784,E2 2214.784} C_VEL
LIN {X 0,Y 575.829,Z 685.03,A -85,B 0,C 180,E1 2220.139,E2 2220.139} C_VEL
LIN {X 0,Y 575.931,Z 685.102,A -85,B 0,C 180,E1 2224.81,E2 2224.81} C_VEL
LIN {X 0,Y 579.161,Z 698.959,A -85,B 0,C 180,E1 2225.519,E2 2225.519} C_VEL
LIN {X 0,Y 578.482,Z 733.694,A -85,B 0,C 180,E1 2227.342,E2 2227.342} C_VEL
LIN {X 0,Y 577.751,Z 766.024,A -85,B 0,C 180,E1 2229.73,E2 2229.73} C_VEL
LIN {X 0,Y 577.04,Z 794.765,A -85,B 0,C 180,E1 2232.591,E2 2232.591} C_VEL
LIN {X 0,Y 576.633,Z 817.506,A -85,B 0,C 180,E1 2235.626,E2 2235.626} C_VEL
LIN {X 0,Y 576.369,Z 835.02,A -85,B 0,C 180,E1 2238.766,E2 2238.766} C_VEL
LIN {X 0,Y 576.257,Z 848.175,A -85,B 0,C 180,E1 2242.098,E2 2242.098} C_VEL
LIN {X 0,Y 576.203,Z 856.565,A -85,B 0,C 180,E1 2245.494,E2 2245.494} C_VEL
LIN {X 0,Y 576.169,Z 860.042,A -85,B 0,C 180,E1 2248.499,E2 2248.499} C_VEL
LIN {X 0,Y 576.25,Z 859.982,A -85,B 0,C 180,E1 2251.501,E2 2251.501} C_VEL
LIN {X 0,Y 576.256,Z 855.208,A -85,B 0,C 180,E1 2255.107,E2 2255.107} C_VEL
LIN {X 0,Y 576.356,Z 845.284,A -85,B 0,C 180,E1 2258.658,E2 2258.658} C_VEL
LIN {X 0,Y 576.471,Z 829.318,A -85,B 0,C 180,E1 2262.28,E2 2262.28} C_VEL
LIN {X 0,Y 576.81,Z 808.76,A -85,B 0,C 180,E1 2265.554,E2 2265.554} C_VEL
LIN {X 0,Y 577.339,Z 784.099,A -85,B 0,C 180,E1 2268.476,E2 2268.476} C_VEL
LIN {X 0,Y 578.04,Z 754.288,A -85,B 0,C 180,E1 2271.135,E2 2271.135} C_VEL
LIN {X 0,Y 578.757,Z 720.812,A -85,B 0,C 180,E1 2273.321,E2 2273.321} C_VEL
LIN {X 0,Y 578.219,Z 693.165,A -85,B 0,C 180,E1 2274.68,E2 2274.68} C_VEL
LIN {X 0,Y 575.995,Z 685.03,A -85,B 0,C 180,E1 2275.169,E2 2275.169} C_VEL
LIN {X 0,Y 575.682,Z 685.03,A -85,B 0,C 180,E1 2280.13,E2 2280.13} C_VEL
LIN {X 0,Y 575.695,Z 685.03,A -85,B 0,C 180,E1 2285.216,E2 2285.216} C_VEL
LIN {X 0,Y 575.631,Z 685.03,A -85,B 0,C 180,E1 2290.947,E2 2290.947} C_VEL
LIN {X 0,Y 575.777,Z 685.03,A -85,B 0,C 180,E1 2297.208,E2 2297.208} C_VEL
LIN {X 0,Y 575.823,Z 685.03,A -85,B 0,C 180,E1 2302.941,E2 2302.941} C_VEL
LIN {X 0,Y 575.7,Z 685.03,A -85,B 0,C 180,E1 2308.39,E2 2308.39} C_VEL
LIN {X 0,Y 575.804,Z 685.03,A -85,B 0,C 180,E1 2313.549,E2 2313.549} C_VEL
LIN {X 0,Y 575.944,Z 685.03,A -85,B 0,C 180,E1 2320.091,E2 2320.091} C_VEL
LIN {X 0,Y 576.151,Z 685.03,A -85,B 0,C 180,E1 2326.37,E2 2326.37} C_VEL
LIN {X 0,Y 575.943,Z 685.03,A -85,B 0,C 180,E1 2332.687,E2 2332.687} C_VEL
LIN {X 0,Y 576.102,Z 685.03,A -85,B 0,C 180,E1 2337,E2 2337} C_VEL
LIN {X 0,Y 576.242,Z 685.03,A -85,B 0,C 180,E1 2341.503,E2 2341.503} C_VEL
LIN {X 0,Y 576.189,Z 685.03,A -85,B 0,C 180,E1 2346.016,E2 2346.016} C_VEL
LIN {X 0,Y 575.839,Z 685.03,A -85,B 0,C 180,E1 2349.158,E2 2349.158} C_VEL
LIN {X 0,Y 571.898,Z 685.03,A -85,B 0,C 180,E1 2350.857,E2 2350.857} C_VEL
LIN {X 0,Y 567.883,Z 685.03,A -85,B 0,C 180,E1 2352.58,E2 2352.58} C_VEL
LIN {X 0,Y 567.915,Z 685.03,A -85,B 0,C 180,E1 2356.996,E2 2356.996} C_VEL
LIN {X 0,Y 567.856,Z 685.03,A -85,B 0,C 180,E1 2361.842,E2 2361.842} C_VEL
LIN {X 0,Y 567.824,Z 685.03,A -85,B 0,C 180,E1 2366.859,E2 2366.859} C_VEL
LIN {X 0,Y 567.668,Z 685.03,A -85,B 0,C 180,E1 2372.118,E2 2372.118} C_VEL
LIN {X 0,Y 567.686,Z 685.03,A -85,B 0,C 180,E1 2377.689,E2 2377.689} C_VEL
LIN {X 0,Y 567.656,Z 685.03,A -85,B 0,C 180,E1 2383.722,E2 2383.722} C_VEL
LIN {X 0,Y 567.776,Z 685.03,A -85,B 0,C 180,E1 2388.361,E2 2388.361} C_VEL
LIN {X 0,Y 568.001,Z 685.03,A -85,B 0,C 180,E1 2394.235,E2 2394.235} C_VEL
LIN {X 0,Y 568.148,Z 685.126,A -85,B 0,C 180,E1 2397.857,E2 2397.857} C_VEL
LIN {X 0,Y 574.287,Z 699.747,A -85,B 0,C 180,E1 2398.452,E2 2398.452} C_VEL
LIN {X 0,Y 574.062,Z 773.325,A -85,B 0,C 180,E1 2399.605,E2 2399.605} C_VEL
LIN {X 0,Y 573.38,Z 810.687,A -85,B 0,C 180,E1 2400.743,E2 2400.743} C_VEL
LIN {X 0,Y 572.387,Z 846.842,A -85,B 0,C 180,E1 2402.42,E2 2402.42} C_VEL
LIN {X 0,Y 571.332,Z 882.111,A -85,B 0,C 180,E1 2404.7,E2 2404.7} C_VEL
LIN {X 0,Y 570.3,Z 914.624,A -85,B 0,C 180,E1 2407.5,E2 2407.5} C_VEL
LIN {X 0,Y 569.418,Z 943.682,A -85,B 0,C 180,E1 2410.776,E2 2410.776} C_VEL
LIN {X 0,Y 568.722,Z 968.077,A -85,B 0,C 180,E1 2414.416,E2 2414.416} C_VEL
LIN {X 0,Y 568.413,Z 986.444,A -85,B 0,C 180,E1 2418.127,E2 2418.127} C_VEL
LIN {X 0,Y 568.32,Z 999.718,A -85,B 0,C 180,E1 2421.987,E2 2421.987} C_VEL
LIN {X 0,Y 568.216,Z 1006.956,A -85,B 0,C 180,E1 2425.43,E2 2425.43} C_VEL
LIN {X 0,Y 568.257,Z 1010.087,A -85,B 0,C 180,E1 2428.478,E2 2428.478} C_VEL
LIN {X 0,Y 568.394,Z 1010.087,A -85,B 0,C 180,E1 2431.521,E2 2431.521} C_VEL
LIN {X 0,Y 568.361,Z 1005.372,A -85,B 0,C 180,E1 2435.53,E2 2435.53} C_VEL
LIN {X 0,Y 568.378,Z 995.072,A -85,B 0,C 180,E1 2439.551,E2 2439.551} C_VEL
LIN {X 0,Y 568.599,Z 979.448,A -85,B 0,C 180,E1 2443.427,E2 2443.427} C_VEL
LIN {X 0,Y 569.032,Z 958.116,A -85,B 0,C 180,E1 2447.194,E2 2447.194} C_VEL
LIN {X 0,Y 569.766,Z 932.871,A -85,B 0,C 180,E1 2450.543,E2 2450.543} C_VEL
LIN {X 0,Y 570.641,Z 903.125,A -85,B 0,C 180,E1 2453.58,E2 2453.58} C_VEL
LIN {X 0,Y 571.755,Z 869.541,A -85,B 0,C 180,E1 2456.192,E2 2456.192} C_VEL
LIN {X 0,Y 572.79,Z 834.346,A -85,B 0,C 180,E1 2458.227,E2 2458.227} C_VEL
LIN {X 0,Y 573.649,Z 797.22,A -85,B 0,C 180,E1 2459.734,E2 2459.734} C_VEL
LIN {X 0,Y 574.352,Z 760.375,A -85,B 0,C 180,E1 2460.65,E2 2460.65} C_VEL
LIN {X 0,Y 573.672,Z 698.23,A -85,B 0,C 180,E1 2461.608,E2 2461.608} C_VEL
LIN {X 0,Y 568.197,Z 685.03,A -85,B 0,C 180,E1 2462.172,E2 2462.172} C_VEL
LIN {X 0,Y 567.937,Z 685.03,A -85,B 0,C 180,E1 2467.669,E2 2467.669} C_VEL
LIN {X 0,Y 567.661,Z 685.03,A -85,B 0,C 180,E1 2473.721,E2 2473.721} C_VEL
LIN {X 0,Y 567.793,Z 685.03,A -85,B 0,C 180,E1 2478.363,E2 2478.363} C_VEL
LIN {X 0,Y 567.955,Z 685.03,A -85,B 0,C 180,E1 2484.231,E2 2484.231} C_VEL
LIN {X 0,Y 567.848,Z 685.03,A -85,B 0,C 180,E1 2489.674,E2 2489.674} C_VEL
LIN {X 0,Y 567.734,Z 685.03,A -85,B 0,C 180,E1 2494.831,E2 2494.831} C_VEL
LIN {X 0,Y 567.79,Z 685.03,A -85,B 0,C 180,E1 2499.786,E2 2499.786} C_VEL
LIN {X 0,Y 567.885,Z 685.03,A -85,B 0,C 180,E1 2504.588,E2 2504.588} C_VEL
LIN {X 0,Y 567.897,Z 685.03,A -85,B 0,C 180,E1 2509.466,E2 2509.466} C_VEL
LIN {X 0,Y 567.972,Z 685.03,A -85,B 0,C 180,E1 2513.897,E2 2513.897} C_VEL
LIN {X 0,Y 567.979,Z 685.03,A -85,B 0,C 180,E1 2518.475,E2 2518.475} C_VEL
LIN {X 0,Y 568.021,Z 685.03,A -85,B 0,C 180,E1 2523.043,E2 2523.043} C_VEL
LIN {X 0,Y 567.942,Z 685.03,A -85,B 0,C 180,E1 2527.631,E2 2527.631} C_VEL
LIN {X 0,Y 567.945,Z 685.03,A -85,B 0,C 180,E1 2532.268,E2 2532.268} C_VEL
LIN {X 0,Y 567.933,Z 685.03,A -85,B 0,C 180,E1 2536.989,E2 2536.989} C_VEL
LIN {X 0,Y 567.878,Z 685.03,A -85,B 0,C 180,E1 2541.835,E2 2541.835} C_VEL
LIN {X 0,Y 567.805,Z 685.03,A -85,B 0,C 180,E1 2546.853,E2 2546.853} C_VEL
LIN {X 0,Y 567.7,Z 685.03,A -85,B 0,C 180,E1 2552.109,E2 2552.109} C_VEL
LIN {X 0,Y 567.882,Z 685.03,A -85,B 0,C 180,E1 2557.667,E2 2557.667} C_VEL
LIN {X 0,Y 567.768,Z 685.03,A -85,B 0,C 180,E1 2563.703,E2 2563.703} C_VEL
LIN {X 0,Y 567.655,Z 685.03,A -85,B 0,C 180,E1 2568.35,E2 2568.35} C_VEL
LIN {X 0,Y 567.725,Z 685.03,A -85,B 0,C 180,E1 2574.215,E2 2574.215} C_VEL
LIN {X 0,Y 567.939,Z 685.03,A -85,B 0,C 180,E1 2579.68,E2 2579.68} C_VEL
LIN {X 0,Y 568.002,Z 685.637,A -85,B 0,C 180,E1 2584.454,E2 2584.454} C_VEL
LIN {X 0,Y 571.889,Z 701.354,A -85,B 0,C 180,E1 2585.292,E2 2585.292} C_VEL
LIN {X 0,Y 571.036,Z 736.065,A -85,B 0,C 180,E1 2587.189,E2 2587.189} C_VEL
LIN {X 0,Y 570.157,Z 767.42,A -85,B 0,C 180,E1 2589.572,E2 2589.572} C_VEL
LIN {X 0,Y 569.305,Z 795.789,A -85,B 0,C 180,E1 2592.468,E2 2592.468} C_VEL
LIN {X 0,Y 568.818,Z 818.677,A -85,B 0,C 180,E1 2595.615,E2 2595.615} C_VEL
LIN {X 0,Y 568.493,Z 836.477,A -85,B 0,C 180,E1 2598.933,E2 2598.933} C_VEL
LIN {X 0,Y 568.331,Z 849.317,A -85,B 0,C 180,E1 2602.371,E2 2602.371} C_VEL
LIN {X 0,Y 568.384,Z 857.76,A -85,B 0,C 180,E1 2606.194,E2 2606.194} C_VEL
LIN {X 0,Y 568.276,Z 860.497,A -85,B 0,C 180,E1 2610,E2 2610} C_VEL
LIN {X 0,Y 568.408,Z 857.618,A -85,B 0,C 180,E1 2613.805,E2 2613.805} C_VEL
LIN {X 0,Y 568.435,Z 849.05,A -85,B 0,C 180,E1 2617.627,E2 2617.627} C_VEL
LIN {X 0,Y 568.608,Z 835.724,A -85,B 0,C 180,E1 2621.143,E2 2621.143} C_VEL
LIN {X 0,Y 568.945,Z 815.749,A -85,B 0,C 180,E1 2624.755,E2 2624.755} C_VEL
LIN {X 0,Y 569.508,Z 791.609,A -85,B 0,C 180,E1 2627.916,E2 2627.916} C_VEL
LIN {X 0,Y 570.278,Z 762.968,A -85,B 0,C 180,E1 2630.727,E2 2630.727} C_VEL
LIN {X 0,Y 571.157,Z 729.846,A -85,B 0,C 180,E1 2633.113,E2 2633.113} C_VEL
LIN {X 0,Y 571.297,Z 696.526,A -85,B 0,C 180,E1 2634.855,E2 2634.855} C_VEL
LIN {X 0,Y 568.075,Z 685.03,A -85,B 0,C 180,E1 2635.556,E2 2635.556} C_VEL
LIN {X 0,Y 567.858,Z 685.03,A -85,B 0,C 180,E1 2641.763,E2 2641.763} C_VEL
LIN {X 0,Y 567.709,Z 685.03,A -85,B 0,C 180,E1 2647.687,E2 2647.687} C_VEL
LIN {X 0,Y 567.697,Z 685.03,A -85,B 0,C 180,E1 2653.718,E2 2653.718} C_VEL
LIN {X 0,Y 567.811,Z 685.03,A -85,B 0,C 180,E1 2658.372,E2 2658.372} C_VEL
LIN {X 0,Y 567.833,Z 685.03,A -85,B 0,C 180,E1 2664.229,E2 2664.229} C_VEL
LIN {X 0,Y 567.796,Z 685.03,A -85,B 0,C 180,E1 2669.678,E2 2669.678} C_VEL
LIN {X 0,Y 567.906,Z 685.03,A -85,B 0,C 180,E1 2674.846,E2 2674.846} C_VEL
LIN {X 0,Y 567.989,Z 685.03,A -85,B 0,C 180,E1 2679.8,E2 2679.8} C_VEL
LIN {X 0,Y 568.228,Z 685.03,A -85,B 0,C 180,E1 2686.176,E2 2686.176} C_VEL
LIN {X 0,Y 568.019,Z 685.03,A -85,B 0,C 180,E1 2692.676,E2 2692.676} C_VEL
LIN {X 0,Y 568.197,Z 685.03,A -85,B 0,C 180,E1 2696.958,E2 2696.958} C_VEL
LIN {X 0,Y 568.355,Z 685.03,A -85,B 0,C 180,E1 2701.524,E2 2701.524} C_VEL
LIN {X 0,Y 568.256,Z 685.03,A -85,B 0,C 180,E1 2706.1,E2 2706.1} C_VEL
LIN {X 0,Y 567.919,Z 685.03,A -85,B 0,C 180,E1 2712.275,E2 2712.275} C_VEL
LIN {X 0,Y 567.883,Z 685.03,A -85,B 0,C 180,E1 2712.58,E2 2712.58} C_VEL
LIN {X 0,Y 563.954,Z 685.03,A -85,B 0,C 180,E1 2714.302,E2 2714.302} C_VEL
LIN {X 0,Y 559.989,Z 685.03,A -85,B 0,C 180,E1 2716.048,E2 2716.048} C_VEL
LIN {X 0,Y 559.907,Z 685.03,A -85,B 0,C 180,E1 2722.169,E2 2722.169} C_VEL
LIN {X 0,Y 559.881,Z 685.03,A -85,B 0,C 180,E1 2727.271,E2 2727.271} C_VEL
LIN {X 0,Y 559.695,Z 685.03,A -85,B 0,C 180,E1 2732.631,E2 2732.631} C_VEL
LIN {X 0,Y 559.834,Z 685.03,A -85,B 0,C 180,E1 2736.37,E2 2736.37} C_VEL
LIN {X 0,Y 559.76,Z 685.03,A -85,B 0,C 180,E1 2742.373,E2 2742.373} C_VEL
LIN {X 0,Y 559.822,Z 685.03,A -85,B 0,C 180,E1 2747.633,E2 2747.633} C_VEL
LIN {X 0,Y 560.077,Z 685.03,A -85,B 0,C 180,E1 2753.927,E2 2753.927} C_VEL
LIN {X 0,Y 560.267,Z 685.171,A -85,B 0,C 180,E1 2757.35,E2 2757.35} C_VEL
LIN {X 0,Y 567.588,Z 704.013,A -85,B 0,C 180,E1 2758.098,E2 2758.098} C_VEL
LIN {X 0,Y 567.214,Z 775.26,A -85,B 0,C 180,E1 2759.242,E2 2759.242} C_VEL
LIN {X 0,Y 566.363,Z 814.345,A -85,B 0,C 180,E1 2760.489,E2 2760.489} C_VEL
LIN {X 0,Y 565.197,Z 852.326,A -85,B 0,C 180,E1 2762.354,E2 2762.354} C_VEL
LIN {X 0,Y 563.804,Z 887.85,A -85,B 0,C 180,E1 2764.788,E2 2764.788} C_VEL
LIN {X 0,Y 562.581,Z 920.094,A -85,B 0,C 180,E1 2767.742,E2 2767.742} C_VEL
LIN {X 0,Y 561.597,Z 947.675,A -85,B 0,C 180,E1 2771.046,E2 2771.046} C_VEL
LIN {X 0,Y 560.923,Z 969.171,A -85,B 0,C 180,E1 2774.394,E2 2774.394} C_VEL
LIN {X 0,Y 560.56,Z 986.443,A -85,B 0,C 180,E1 2777.958,E2 2777.958} C_VEL
LIN {X 0,Y 560.458,Z 999.718,A -85,B 0,C 180,E1 2781.874,E2 2781.874} C_VEL
LIN {X 0,Y 560.322,Z 1006.957,A -85,B 0,C 180,E1 2785.366,E2 2785.366} C_VEL
LIN {X 0,Y 560.356,Z 1010.087,A -85,B 0,C 180,E1 2788.457,E2 2788.457} C_VEL
LIN {X 0,Y 560.487,Z 1010.087,A -85,B 0,C 180,E1 2791.543,E2 2791.543} C_VEL
LIN {X 0,Y 560.48,Z 1005.831,A -85,B 0,C 180,E1 2795.36,E2 2795.36} C_VEL
LIN {X 0,Y 560.522,Z 996.303,A -85,B 0,C 180,E1 2799.296,E2 2799.296} C_VEL
LIN {X 0,Y 560.773,Z 981.282,A -85,B 0,C 180,E1 2803.222,E2 2803.222} C_VEL
LIN {X 0,Y 561.216,Z 960.92,A -85,B 0,C 180,E1 2807.002,E2 2807.002} C_VEL
LIN {X 0,Y 562.087,Z 934.616,A -85,B 0,C 180,E1 2810.632,E2 2810.632} C_VEL
LIN {X 0,Y 563.197,Z 903.987,A -85,B 0,C 180,E1 2813.832,E2 2813.832} C_VEL
LIN {X 0,Y 564.441,Z 871.019,A -85,B 0,C 180,E1 2816.453,E2 2816.453} C_VEL
LIN {X 0,Y 565.666,Z 836.178,A -85,B 0,C 180,E1 2818.521,E2 2818.521} C_VEL
LIN {X 0,Y 566.703,Z 799.21,A -85,B 0,C 180,E1 2820.068,E2 2820.068} C_VEL
LIN {X 0,Y 567.536,Z 761.609,A -85,B 0,C 180,E1 2821.038,E2 2821.038} C_VEL
LIN {X 0,Y 567.145,Z 701.338,A -85,B 0,C 180,E1 2821.969,E2 2821.969} C_VEL
LIN {X 0,Y 560.339,Z 685.03,A -85,B 0,C 180,E1 2822.686,E2 2822.686} C_VEL
LIN {X 0,Y 559.9,Z 685.03,A -85,B 0,C 180,E1 2828.595,E2 2828.595} C_VEL
LIN {X 0,Y 559.699,Z 685.03,A -85,B 0,C 180,E1 2834.506,E2 2834.506} C_VEL
LIN {X 0,Y 559.83,Z 685.03,A -85,B 0,C 180,E1 2839.691,E2 2839.691} C_VEL
LIN {X 0,Y 560.044,Z 685.03,A -85,B 0,C 180,E1 2845.54,E2 2845.54} C_VEL
LIN {X 0,Y 559.882,Z 685.03,A -85,B 0,C 180,E1 2850.978,E2 2850.978} C_VEL
LIN {X 0,Y 559.9,Z 685.03,A -85,B 0,C 180,E1 2856.396,E2 2856.396} C_VEL
LIN {X 0,Y 560.07,Z 685.03,A -85,B 0,C 180,E1 2862.758,E2 2862.758} C_VEL
LIN {X 0,Y 560.094,Z 685.03,A -85,B 0,C 180,E1 2867.551,E2 2867.551} C_VEL
LIN {X 0,Y 560.141,Z 685.03,A -85,B 0,C 180,E1 2872.256,E2 2872.256} C_VEL
LIN {X 0,Y 560.313,Z 685.03,A -85,B 0,C 180,E1 2876.91,E2 2876.91} C_VEL
LIN {X 0,Y 560.431,Z 685.03,A -85,B 0,C 180,E1 2881.54,E2 2881.54} C_VEL
LIN {X 0,Y 560.359,Z 685.03,A -85,B 0,C 180,E1 2886.18,E2 2886.18} C_VEL
LIN {X 0,Y 560.025,Z 685.03,A -85,B 0,C 180,E1 2892.444,E2 2892.444} C_VEL
LIN {X 0,Y 559.999,Z 685.03,A -85,B 0,C 180,E1 2897.238,E2 2897.238} C_VEL
LIN {X 0,Y 559.929,Z 685.03,A -85,B 0,C 180,E1 2902.161,E2 2902.161} C_VEL
LIN {X 0,Y 559.858,Z 685.03,A -85,B 0,C 180,E1 2907.266,E2 2907.266} C_VEL
LIN {X 0,Y 559.728,Z 685.03,A -85,B 0,C 180,E1 2912.622,E2 2912.622} C_VEL
LIN {X 0,Y 559.892,Z 685.03,A -85,B 0,C 180,E1 2918.301,E2 2918.301} C_VEL
LIN {X 0,Y 559.827,Z 685.03,A -85,B 0,C 180,E1 2923.3,E2 2923.3} C_VEL
LIN {X 0,Y 559.731,Z 685.03,A -85,B 0,C 180,E1 2929.004,E2 2929.004} C_VEL
LIN {X 0,Y 559.815,Z 685.03,A -85,B 0,C 180,E1 2933.954,E2 2933.954} C_VEL
LIN {X 0,Y 560.04,Z 685.03,A -85,B 0,C 180,E1 2939.554,E2 2939.554} C_VEL
LIN {X 0,Y 560.053,Z 685.4,A -85,B 0,C 180,E1 2944.056,E2 2944.056} C_VEL
LIN {X 0,Y 564.577,Z 703.878,A -85,B 0,C 180,E1 2945.074,E2 2945.074} C_VEL
LIN {X 0,Y 563.573,Z 737.698,A -85,B 0,C 180,E1 2946.982,E2 2946.982} C_VEL
LIN {X 0,Y 562.583,Z 768.553,A -85,B 0,C 180,E1 2949.388,E2 2949.388} C_VEL
LIN {X 0,Y 561.599,Z 796.69,A -85,B 0,C 180,E1 2952.334,E2 2952.334} C_VEL
LIN {X 0,Y 560.979,Z 820.174,A -85,B 0,C 180,E1 2955.657,E2 2955.657} C_VEL
LIN {X 0,Y 560.612,Z 838.085,A -85,B 0,C 180,E1 2959.14,E2 2959.14} C_VEL
LIN {X 0,Y 560.468,Z 850.458,A -85,B 0,C 180,E1 2962.652,E2 2962.652} C_VEL
LIN {X 0,Y 560.492,Z 857.76,A -85,B 0,C 180,E1 2966.141,E2 2966.141} C_VEL
LIN {X 0,Y 560.377,Z 860.497,A -85,B 0,C 180,E1 2970,E2 2970} C_VEL
LIN {X 0,Y 560.518,Z 857.619,A -85,B 0,C 180,E1 2973.859,E2 2973.859} C_VEL
LIN {X 0,Y 560.551,Z 849.052,A -85,B 0,C 180,E1 2977.735,E2 2977.735} C_VEL
LIN {X 0,Y 560.736,Z 835.423,A -85,B 0,C 180,E1 2981.37,E2 2981.37} C_VEL
LIN {X 0,Y 561.173,Z 815.596,A -85,B 0,C 180,E1 2984.987,E2 2984.987} C_VEL
LIN {X 0,Y 561.867,Z 790.925,A -85,B 0,C 180,E1 2988.248,E2 2988.248} C_VEL
LIN {X 0,Y 562.774,Z 761.802,A -85,B 0,C 180,E1 2991.119,E2 2991.119} C_VEL
LIN {X 0,Y 563.793,Z 729.273,A -85,B 0,C 180,E1 2993.469,E2 2993.469} C_VEL
LIN {X 0,Y 564.094,Z 698.931,A -85,B 0,C 180,E1 2995.089,E2 2995.089} C_VEL
LIN {X 0,Y 560.136,Z 685.03,A -85,B 0,C 180,E1 2995.905,E2 2995.905} C_VEL
LIN {X 0,Y 559.877,Z 685.03,A -85,B 0,C 180,E1 3000.803,E2 3000.803} C_VEL
LIN {X 0,Y 559.803,Z 685.03,A -85,B 0,C 180,E1 3006.372,E2 3006.372} C_VEL
LIN {X 0,Y 559.748,Z 685.03,A -85,B 0,C 180,E1 3012.373,E2 3012.373} C_VEL
LIN {X 0,Y 559.868,Z 685.03,A -85,B 0,C 180,E1 3017.646,E2 3017.646} C_VEL
LIN {X 0,Y 559.948,Z 685.03,A -85,B 0,C 180,E1 3023.946,E2 3023.946} C_VEL
LIN {X 0,Y 559.903,Z 685.03,A -85,B 0,C 180,E1 3029.591,E2 3029.591} C_VEL
LIN {X 0,Y 559.982,Z 685.03,A -85,B 0,C 180,E1 3034.464,E2 3034.464} C_VEL
LIN {X 0,Y 560.06,Z 685.03,A -85,B 0,C 180,E1 3040.565,E2 3040.565} C_VEL
LIN {X 0,Y 560.277,Z 685.03,A -85,B 0,C 180,E1 3045.976,E2 3045.976} C_VEL
LIN {X 0,Y 560.107,Z 685.03,A -85,B 0,C 180,E1 3052.666,E2 3052.666} C_VEL
LIN {X 0,Y 560.288,Z 685.03,A -85,B 0,C 180,E1 3056.915,E2 3056.915} C_VEL
LIN {X 0,Y 560.444,Z 685.03,A -85,B 0,C 180,E1 3061.546,E2 3061.546} C_VEL
LIN {X 0,Y 560.345,Z 685.03,A -85,B 0,C 180,E1 3066.186,E2 3066.186} C_VEL
LIN {X 0,Y 559.983,Z 685.03,A -85,B 0,C 180,E1 3072.572,E2 3072.572} C_VEL
LIN {X 0,Y 559.989,Z 685.03,A -85,B 0,C 180,E1 3076.048,E2 3076.048} C_VEL
LIN {X 0,Y 555.987,Z 685.03,A -85,B 0,C 180,E1 3077.792,E2 3077.792} C_VEL
LIN {X 0,Y 552.001,Z 685.03,A -85,B 0,C 180,E1 3079.56,E2 3079.56} C_VEL
LIN {X 0,Y 552.054,Z 685.03,A -85,B 0,C 180,E1 3085.574,E2 3085.574} C_VEL
LIN {X 0,Y 551.823,Z 685.03,A -85,B 0,C 180,E1 3091.304,E2 3091.304} C_VEL
LIN {X 0,Y 551.822,Z 685.03,A -85,B 0,C 180,E1 3096.985,E2 3096.985} C_VEL
LIN {X 0,Y 551.813,Z 685.03,A -85,B 0,C 180,E1 3103.13,E2 3103.13} C_VEL
LIN {X 0,Y 551.952,Z 685.03,A -85,B 0,C 180,E1 3108.994,E2 3108.994} C_VEL
LIN {X 0,Y 552.165,Z 685.03,A -85,B 0,C 180,E1 3115.07,E2 3115.07} C_VEL
LIN {X 0,Y 552.33,Z 685.166,A -85,B 0,C 180,E1 3116.821,E2 3116.821} C_VEL
LIN {X 0,Y 560.879,Z 706.152,A -85,B 0,C 180,E1 3117.702,E2 3117.702} C_VEL
LIN {X 0,Y 560.41,Z 775.26,A -85,B 0,C 180,E1 3118.827,E2 3118.827} C_VEL
LIN {X 0,Y 559.431,Z 814.276,A -85,B 0,C 180,E1 3120.084,E2 3120.084} C_VEL
LIN {X 0,Y 558.043,Z 852.197,A -85,B 0,C 180,E1 3121.961,E2 3121.961} C_VEL
LIN {X 0,Y 556.42,Z 888.982,A -85,B 0,C 180,E1 3124.526,E2 3124.526} C_VEL
LIN {X 0,Y 555.088,Z 920.236,A -85,B 0,C 180,E1 3127.441,E2 3127.441} C_VEL
LIN {X 0,Y 553.912,Z 946.91,A -85,B 0,C 180,E1 3130.665,E2 3130.665} C_VEL
LIN {X 0,Y 553.093,Z 969.172,A -85,B 0,C 180,E1 3134.167,E2 3134.167} C_VEL
LIN {X 0,Y 552.716,Z 986.444,A -85,B 0,C 180,E1 3137.785,E2 3137.785} C_VEL
LIN {X 0,Y 552.594,Z 999.718,A -85,B 0,C 180,E1 3141.757,E2 3141.757} C_VEL
LIN {X 0,Y 552.453,Z 1006.957,A -85,B 0,C 180,E1 3145.3,E2 3145.3} C_VEL
LIN {X 0,Y 552.461,Z 1010.087,A -85,B 0,C 180,E1 3148.435,E2 3148.435} C_VEL
LIN {X 0,Y 552.581,Z 1010.087,A -85,B 0,C 180,E1 3151.565,E2 3151.565} C_VEL
LIN {X 0,Y 552.565,Z 1005.756,A -85,B 0,C 180,E1 3155.485,E2 3155.485} C_VEL
LIN {X 0,Y 552.623,Z 996.303,A -85,B 0,C 180,E1 3159.43,E2 3159.43} C_VEL
LIN {X 0,Y 552.921,Z 981.282,A -85,B 0,C 180,E1 3163.413,E2 3163.413} C_VEL
LIN {X 0,Y 553.518,Z 959.669,A -85,B 0,C 180,E1 3167.45,E2 3167.45} C_VEL
LIN {X 0,Y 554.475,Z 934.615,A -85,B 0,C 180,E1 3170.928,E2 3170.928} C_VEL
LIN {X 0,Y 555.771,Z 903.988,A -85,B 0,C 180,E1 3174.17,E2 3174.17} C_VEL
LIN {X 0,Y 557.19,Z 871.713,A -85,B 0,C 180,E1 3176.775,E2 3176.775} C_VEL
LIN {X 0,Y 558.614,Z 836.668,A -85,B 0,C 180,E1 3178.889,E2 3178.889} C_VEL
LIN {X 0,Y 559.829,Z 799.834,A -85,B 0,C 180,E1 3180.455,E2 3180.455} C_VEL
LIN {X 0,Y 560.78,Z 761.609,A -85,B 0,C 180,E1 3181.454,E2 3181.454} C_VEL
LIN {X 0,Y 560.435,Z 703.66,A -85,B 0,C 180,E1 3182.364,E2 3182.364} C_VEL
LIN {X 0,Y 552.366,Z 685.03,A -85,B 0,C 180,E1 3183.212,E2 3183.212} C_VEL
LIN {X 0,Y 551.964,Z 685.03,A -85,B 0,C 180,E1 3188.961,E2 3188.961} C_VEL
LIN {X 0,Y 551.809,Z 685.03,A -85,B 0,C 180,E1 3194.683,E2 3194.683} C_VEL
LIN {X 0,Y 551.924,Z 685.03,A -85,B 0,C 180,E1 3199.955,E2 3199.955} C_VEL
LIN {X 0,Y 552.128,Z 685.03,A -85,B 0,C 180,E1 3205.076,E2 3205.076} C_VEL
LIN {X 0,Y 552.001,Z 685.03,A -85,B 0,C 180,E1 3211.018,E2 3211.018} C_VEL
LIN {X 0,Y 551.911,Z 685.03,A -85,B 0,C 180,E1 3215.786,E2 3215.786} C_VEL
LIN {X 0,Y 552.086,Z 685.03,A -85,B 0,C 180,E1 3220.851,E2 3220.851} C_VEL
LIN {X 0,Y 552.213,Z 685.03,A -85,B 0,C 180,E1 3225.761,E2 3225.761} C_VEL
LIN {X 0,Y 552.224,Z 685.03,A -85,B 0,C 180,E1 3232.145,E2 3232.145} C_VEL
LIN {X 0,Y 552.412,Z 685.03,A -85,B 0,C 180,E1 3236.865,E2 3236.865} C_VEL
LIN {X 0,Y 552.524,Z 685.03,A -85,B 0,C 180,E1 3241.562,E2 3241.562} C_VEL
LIN {X 0,Y 552.427,Z 685.03,A -85,B 0,C 180,E1 3246.269,E2 3246.269} C_VEL
LIN {X 0,Y 552.115,Z 685.03,A -85,B 0,C 180,E1 3252.626,E2 3252.626} C_VEL
LIN {X 0,Y 552.087,Z 685.03,A -85,B 0,C 180,E1 3257.493,E2 3257.493} C_VEL
LIN {X 0,Y 551.993,Z 685.03,A -85,B 0,C 180,E1 3262.497,E2 3262.497} C_VEL
LIN {X 0,Y 551.895,Z 685.03,A -85,B 0,C 180,E1 3267.693,E2 3267.693} C_VEL
LIN {X 0,Y 551.822,Z 685.03,A -85,B 0,C 180,E1 3273.149,E2 3273.149} C_VEL
LIN {X 0,Y 551.949,Z 685.03,A -85,B 0,C 180,E1 3278.955,E2 3278.955} C_VEL
LIN {X 0,Y 551.89,Z 685.03,A -85,B 0,C 180,E1 3284.692,E2 3284.692} C_VEL
LIN {X 0,Y 551.813,Z 685.03,A -85,B 0,C 180,E1 3289.959,E2 3289.959} C_VEL
LIN {X 0,Y 551.976,Z 685.03,A -85,B 0,C 180,E1 3295.088,E2 3295.088} C_VEL
LIN {X 0,Y 552.104,Z 685.03,A -85,B 0,C 180,E1 3300.986,E2 3300.986} C_VEL
LIN {X 0,Y 552.145,Z 685.032,A -85,B 0,C 180,E1 3303.643,E2 3303.643} C_VEL
LIN {X 0,Y 557.28,Z 706.215,A -85,B 0,C 180,E1 3304.843,E2 3304.843} C_VEL
LIN {X 0,Y 556.132,Z 739.462,A -85,B 0,C 180,E1 3306.779,E2 3306.779} C_VEL
LIN {X 0,Y 554.955,Z 770.816,A -85,B 0,C 180,E1 3309.299,E2 3309.299} C_VEL
LIN {X 0,Y 553.861,Z 797.859,A -85,B 0,C 180,E1 3312.229,E2 3312.229} C_VEL
LIN {X 0,Y 553.157,Z 820.75,A -85,B 0,C 180,E1 3315.547,E2 3315.547} C_VEL
LIN {X 0,Y 552.739,Z 838.081,A -85,B 0,C 180,E1 3318.983,E2 3318.983} C_VEL
LIN {X 0,Y 552.571,Z 850.457,A -85,B 0,C 180,E1 3322.547,E2 3322.547} C_VEL
LIN {X 0,Y 552.601,Z 857.759,A -85,B 0,C 180,E1 3326.086,E2 3326.086} C_VEL
LIN {X 0,Y 552.477,Z 860.497,A -85,B 0,C 180,E1 3330,E2 3330} C_VEL
LIN {X 0,Y 552.629,Z 857.621,A -85,B 0,C 180,E1 3333.914,E2 3333.914} C_VEL
LIN {X 0,Y 552.67,Z 849.054,A -85,B 0,C 180,E1 3337.846,E2 3337.846} C_VEL
LIN {X 0,Y 552.865,Z 835.956,A -85,B 0,C 180,E1 3341.413,E2 3341.413} C_VEL
LIN {X 0,Y 553.377,Z 816.886,A -85,B 0,C 180,E1 3345.004,E2 3345.004} C_VEL
LIN {X 0,Y 554.118,Z 793.163,A -85,B 0,C 180,E1 3348.25,E2 3348.25} C_VEL
LIN {X 0,Y 555.14,Z 765.271,A -85,B 0,C 180,E1 3351.11,E2 3351.11} C_VEL
LIN {X 0,Y 556.362,Z 732.371,A -85,B 0,C 180,E1 3353.607,E2 3353.607} C_VEL
LIN {X 0,Y 556.816,Z 701.021,A -85,B 0,C 180,E1 3355.348,E2 3355.348} C_VEL
LIN {X 0,Y 552.223,Z 685.03,A -85,B 0,C 180,E1 3356.356,E2 3356.356} C_VEL
LIN {X 0,Y 551.965,Z 685.03,A -85,B 0,C 180,E1 3362.072,E2 3362.072} C_VEL
LIN {X 0,Y 551.822,Z 685.03,A -85,B 0,C 180,E1 3367.541,E2 3367.541} C_VEL
LIN {X 0,Y 551.853,Z 685.03,A -85,B 0,C 180,E1 3373.126,E2 3373.126} C_VEL
LIN {X 0,Y 551.977,Z 685.03,A -85,B 0,C 180,E1 3379.004,E2 3379.004} C_VEL
LIN {X 0,Y 551.93,Z 685.03,A -85,B 0,C 180,E1 3385.106,E2 3385.106} C_VEL
LIN {X 0,Y 551.93,Z 685.03,A -85,B 0,C 180,E1 3391.032,E2 3391.032} C_VEL
LIN {X 0,Y 551.993,Z 685.03,A -85,B 0,C 180,E1 3395.797,E2 3395.797} C_VEL
LIN {X 0,Y 552.179,Z 685.03,A -85,B 0,C 180,E1 3400.861,E2 3400.861} C_VEL
LIN {X 0,Y 552.362,Z 685.03,A -85,B 0,C 180,E1 3405.771,E2 3405.771} C_VEL
LIN {X 0,Y 552.255,Z 685.03,A -85,B 0,C 180,E1 3412.151,E2 3412.151} C_VEL
LIN {X 0,Y 552.388,Z 685.03,A -85,B 0,C 180,E1 3416.871,E2 3416.871} C_VEL
LIN {X 0,Y 552.535,Z 685.03,A -85,B 0,C 180,E1 3421.568,E2 3421.568} C_VEL
LIN {X 0,Y 552.414,Z 685.03,A -85,B 0,C 180,E1 3426.276,E2 3426.276} C_VEL
LIN {X 0,Y 552.087,Z 685.03,A -85,B 0,C 180,E1 3432.632,E2 3432.632} C_VEL
LIN {X 0,Y 552.067,Z 685.03,A -85,B 0,C 180,E1 3437.5,E2 3437.5} C_VEL
LIN {X 0,Y 552.001,Z 685.03,A -85,B 0,C 180,E1 3439.56,E2 3439.56} C_VEL
LIN {X 0,Y 547.999,Z 685.03,A -85,B 0,C 180,E1 3441.331,E2 3441.331} C_VEL
LIN {X 0,Y 544.012,Z 685.03,A -85,B 0,C 180,E1 3443.127,E2 3443.127} C_VEL
LIN {X 0,Y 543.982,Z 685.03,A -85,B 0,C 180,E1 3448.138,E2 3448.138} C_VEL
LIN {X 0,Y 543.868,Z 685.03,A -85,B 0,C 180,E1 3453.705,E2 3453.705} C_VEL
LIN {X 0,Y 543.851,Z 685.03,A -85,B 0,C 180,E1 3459.656,E2 3459.656} C_VEL
LIN {X 0,Y 543.861,Z 685.03,A -85,B 0,C 180,E1 3463.92,E2 3463.92} C_VEL
LIN {X 0,Y 544.013,Z 685.03,A -85,B 0,C 180,E1 3470.359,E2 3470.359} C_VEL
LIN {X 0,Y 544.345,Z 685.03,A -85,B 0,C 180,E1 3476.266,E2 3476.266} C_VEL
LIN {X 0,Y 554.22,Z 707.61,A -85,B 0,C 180,E1 3477.288,E2 3477.288} C_VEL
LIN {X 0,Y 553.652,Z 775.119,A -85,B 0,C 180,E1 3478.4,E2 3478.4} C_VEL
LIN {X 0,Y 552.515,Z 814.445,A -85,B 0,C 180,E1 3479.677,E2 3479.677} C_VEL
LIN {X 0,Y 550.892,Z 853.211,A -85,B 0,C 180,E1 3481.628,E2 3481.628} C_VEL
LIN {X 0,Y 549.175,Z 888.329,A -85,B 0,C 180,E1 3484.109,E2 3484.109} C_VEL
LIN {X 0,Y 547.568,Z 920.04,A -85,B 0,C 180,E1 3487.092,E2 3487.092} C_VEL
LIN {X 0,Y 546.227,Z 947.331,A -85,B 0,C 180,E1 3490.442,E2 3490.442} C_VEL
LIN {X 0,Y 545.29,Z 970.265,A -85,B 0,C 180,E1 3494.141,E2 3494.141} C_VEL
LIN {X 0,Y 544.825,Z 987.982,A -85,B 0,C 180,E1 3498.011,E2 3498.011} C_VEL
LIN {X 0,Y 544.715,Z 999.718,A -85,B 0,C 180,E1 3501.637,E2 3501.637} C_VEL
LIN {X 0,Y 544.553,Z 1006.957,A -85,B 0,C 180,E1 3505.231,E2 3505.231} C_VEL
LIN {X 0,Y 544.56,Z 1010.087,A -85,B 0,C 180,E1 3508.412,E2 3508.412} C_VEL
LIN {X 0,Y 544.675,Z 1010.087,A -85,B 0,C 180,E1 3511.588,E2 3511.588} C_VEL
LIN {X 0,Y 544.663,Z 1005.756,A -85,B 0,C 180,E1 3515.565,E2 3515.565} C_VEL
LIN {X 0,Y 544.725,Z 996.303,A -85,B 0,C 180,E1 3519.568,E2 3519.568} C_VEL
LIN {X 0,Y 545.068,Z 981.441,A -85,B 0,C 180,E1 3523.573,E2 3523.573} C_VEL
LIN {X 0,Y 545.729,Z 960.795,A -85,B 0,C 180,E1 3527.522,E2 3527.522} C_VEL
LIN {X 0,Y 546.866,Z 934.745,A -85,B 0,C 180,E1 3531.217,E2 3531.217} C_VEL
LIN {X 0,Y 548.342,Z 904.265,A -85,B 0,C 180,E1 3534.493,E2 3534.493} C_VEL
LIN {X 0,Y 550.002,Z 870.984,A -85,B 0,C 180,E1 3537.207,E2 3537.207} C_VEL
LIN {X 0,Y 551.662,Z 836.324,A -85,B 0,C 180,E1 3539.307,E2 3539.307} C_VEL
LIN {X 0,Y 552.943,Z 800.338,A -85,B 0,C 180,E1 3540.858,E2 3540.858} C_VEL
LIN {X 0,Y 554.04,Z 763.213,A -85,B 0,C 180,E1 3541.852,E2 3541.852} C_VEL
LIN {X 0,Y 553.541,Z 705.797,A -85,B 0,C 180,E1 3542.785,E2 3542.785} C_VEL
LIN {X 0,Y 544.395,Z 685.03,A -85,B 0,C 180,E1 3543.741,E2 3543.741} C_VEL
LIN {X 0,Y 544.013,Z 685.03,A -85,B 0,C 180,E1 3549.641,E2 3549.641} C_VEL
LIN {X 0,Y 543.929,Z 685.03,A -85,B 0,C 180,E1 3556.162,E2 3556.162} C_VEL
LIN {X 0,Y 544.114,Z 685.03,A -85,B 0,C 180,E1 3562.401,E2 3562.401} C_VEL
LIN {X 0,Y 544.13,Z 685.03,A -85,B 0,C 180,E1 3568.202,E2 3568.202} C_VEL
LIN {X 0,Y 543.947,Z 685.03,A -85,B 0,C 180,E1 3573.648,E2 3573.648} C_VEL
LIN {X 0,Y 544.026,Z 685.03,A -85,B 0,C 180,E1 3578.862,E2 3578.862} C_VEL
LIN {X 0,Y 544.181,Z 685.03,A -85,B 0,C 180,E1 3583.899,E2 3583.899} C_VEL
LIN {X 0,Y 544.181,Z 685.03,A -85,B 0,C 180,E1 3588.805,E2 3588.805} C_VEL
LIN {X 0,Y 544.298,Z 685.03,A -85,B 0,C 180,E1 3593.631,E2 3593.631} C_VEL
LIN {X 0,Y 544.301,Z 685.03,A -85,B 0,C 180,E1 3598.408,E2 3598.408} C_VEL
LIN {X 0,Y 544.324,Z 685.03,A -85,B 0,C 180,E1 3603.175,E2 3603.175} C_VEL
LIN {X 0,Y 544.222,Z 685.03,A -85,B 0,C 180,E1 3607.965,E2 3607.965} C_VEL
LIN {X 0,Y 544.197,Z 685.03,A -85,B 0,C 180,E1 3612.812,E2 3612.812} C_VEL
LIN {X 0,Y 544.155,Z 685.03,A -85,B 0,C 180,E1 3617.756,E2 3617.756} C_VEL
LIN {X 0,Y 544.061,Z 685.03,A -85,B 0,C 180,E1 3623.755,E2 3623.755} C_VEL
LIN {X 0,Y 543.966,Z 685.03,A -85,B 0,C 180,E1 3628.132,E2 3628.132} C_VEL
LIN {X 0,Y 543.893,Z 685.03,A -85,B 0,C 180,E1 3633.696,E2 3633.696} C_VEL
LIN {X 0,Y 544.014,Z 685.03,A -85,B 0,C 180,E1 3639.634,E2 3639.634} C_VEL
LIN {X 0,Y 543.977,Z 685.03,A -85,B 0,C 180,E1 3643.9,E2 3643.9} C_VEL
LIN {X 0,Y 543.895,Z 685.03,A -85,B 0,C 180,E1 3650.349,E2 3650.349} C_VEL
LIN {X 0,Y 544.096,Z 685.03,A -85,B 0,C 180,E1 3656.311,E2 3656.311} C_VEL
LIN {X 0,Y 544.163,Z 685.03,A -85,B 0,C 180,E1 3662.531,E2 3662.531} C_VEL
LIN {X 0,Y 544.276,Z 685.929,A -85,B 0,C 180,E1 3663.268,E2 3663.268} C_VEL
LIN {X 0,Y 549.976,Z 707.813,A -85,B 0,C 180,E1 3664.567,E2 3664.567} C_VEL
LIN {X 0,Y 548.616,Z 742.184,A -85,B 0,C 180,E1 3666.635,E2 3666.635} C_VEL
LIN {X 0,Y 547.226,Z 774.011,A -85,B 0,C 180,E1 3669.315,E2 3669.315} C_VEL
LIN {X 0,Y 546.078,Z 800.444,A -85,B 0,C 180,E1 3672.304,E2 3672.304} C_VEL
LIN {X 0,Y 545.309,Z 822.865,A -85,B 0,C 180,E1 3675.696,E2 3675.696} C_VEL
LIN {X 0,Y 544.888,Z 840.133,A -85,B 0,C 180,E1 3679.328,E2 3679.328} C_VEL
LIN {X 0,Y 544.706,Z 851.508,A -85,B 0,C 180,E1 3682.839,E2 3682.839} C_VEL
LIN {X 0,Y 544.712,Z 858.729,A -85,B 0,C 180,E1 3686.824,E2 3686.824} C_VEL
LIN {X 0,Y 544.577,Z 860.497,A -85,B 0,C 180,E1 3690,E2 3690} C_VEL
LIN {X 0,Y 544.632,Z 858.631,A -85,B 0,C 180,E1 3693.177,E2 3693.177} C_VEL
LIN {X 0,Y 544.73,Z 851.295,A -85,B 0,C 180,E1 3697.161,E2 3697.161} C_VEL
LIN {X 0,Y 544.987,Z 837.693,A -85,B 0,C 180,E1 3701.176,E2 3701.176} C_VEL
LIN {X 0,Y 545.502,Z 819.496,A -85,B 0,C 180,E1 3704.784,E2 3704.784} C_VEL
LIN {X 0,Y 546.323,Z 796.559,A -85,B 0,C 180,E1 3708.104,E2 3708.104} C_VEL
LIN {X 0,Y 547.433,Z 768.706,A -85,B 0,C 180,E1 3711.104,E2 3711.104} C_VEL
LIN {X 0,Y 548.784,Z 737.399,A -85,B 0,C 180,E1 3713.605,E2 3713.605} C_VEL
LIN {X 0,Y 549.434,Z 702.848,A -85,B 0,C 180,E1 3715.623,E2 3715.623} C_VEL
LIN {X 0,Y 544.26,Z 685.03,A -85,B 0,C 180,E1 3716.759,E2 3716.759} C_VEL
LIN {X 0,Y 544.063,Z 685.03,A -85,B 0,C 180,E1 3721.801,E2 3721.801} C_VEL
LIN {X 0,Y 543.938,Z 685.03,A -85,B 0,C 180,E1 3727.613,E2 3727.613} C_VEL
LIN {X 0,Y 543.921,Z 685.03,A -85,B 0,C 180,E1 3733.913,E2 3733.913} C_VEL
LIN {X 0,Y 544.038,Z 685.03,A -85,B 0,C 180,E1 3738.495,E2 3738.495} C_VEL
LIN {X 0,Y 543.979,Z 685.03,A -85,B 0,C 180,E1 3744.377,E2 3744.377} C_VEL
LIN {X 0,Y 543.962,Z 685.03,A -85,B 0,C 180,E1 3750.05,E2 3750.05} C_VEL
LIN {X 0,Y 544.091,Z 685.03,A -85,B 0,C 180,E1 3755.422,E2 3755.422} C_VEL
LIN {X 0,Y 544.236,Z 685.03,A -85,B 0,C 180,E1 3760.571,E2 3760.571} C_VEL
LIN {X 0,Y 544.43,Z 685.03,A -85,B 0,C 180,E1 3765.952,E2 3765.952} C_VEL
LIN {X 0,Y 544.339,Z 685.03,A -85,B 0,C 180,E1 3772.036,E2 3772.036} C_VEL
LIN {X 0,Y 544.48,Z 685.03,A -85,B 0,C 180,E1 3776.826,E2 3776.826} C_VEL
LIN {X 0,Y 544.624,Z 685.03,A -85,B 0,C 180,E1 3781.591,E2 3781.591} C_VEL
LIN {X 0,Y 544.488,Z 685.03,A -85,B 0,C 180,E1 3786.367,E2 3786.367} C_VEL
LIN {X 0,Y 544.169,Z 685.03,A -85,B 0,C 180,E1 3792.819,E2 3792.819} C_VEL
LIN {X 0,Y 544.133,Z 685.03,A -85,B 0,C 180,E1 3797.763,E2 3797.763} C_VEL
LIN {X 0,Y 544.012,Z 685.03,A -85,B 0,C 180,E1 3803.127,E2 3803.127} C_VEL
LIN {X 0,Y 542.722,Z 685.03,A -85,B 0,C 180,E1 3804.039,E2 3804.039} C_VEL
LIN {X 0,Y 536.164,Z 685.03,A -85,B 0,C 180,E1 3806.524,E2 3806.524} C_VEL
LIN {X 0,Y 536.092,Z 685.03,A -85,B 0,C 180,E1 3806.76,E2 3806.76} C_VEL
LIN {X 0,Y 535.955,Z 685.03,A -85,B 0,C 180,E1 3812.365,E2 3812.365} C_VEL
LIN {X 0,Y 535.94,Z 685.03,A -85,B 0,C 180,E1 3818.275,E2 3818.275} C_VEL
LIN {X 0,Y 535.893,Z 685.03,A -85,B 0,C 180,E1 3824.746,E2 3824.746} C_VEL
LIN {X 0,Y 536.045,Z 685.03,A -85,B 0,C 180,E1 3829.65,E2 3829.65} C_VEL
LIN {X 0,Y 536.336,Z 685.308,A -85,B 0,C 180,E1 3835.699,E2 3835.699} C_VEL
LIN {X 0,Y 547.437,Z 709.635,A -85,B 0,C 180,E1 3836.862,E2 3836.862} C_VEL
LIN {X 0,Y 546.865,Z 776.987,A -85,B 0,C 180,E1 3838.008,E2 3838.008} C_VEL
LIN {X 0,Y 545.597,Z 815.906,A -85,B 0,C 180,E1 3839.314,E2 3839.314} C_VEL
LIN {X 0,Y 543.788,Z 852.907,A -85,B 0,C 180,E1 3841.203,E2 3841.203} C_VEL
LIN {X 0,Y 541.858,Z 888.659,A -85,B 0,C 180,E1 3843.762,E2 3843.762} C_VEL
LIN {X 0,Y 540.095,Z 920.04,A -85,B 0,C 180,E1 3846.756,E2 3846.756} C_VEL
LIN {X 0,Y 538.595,Z 947.333,A -85,B 0,C 180,E1 3850.153,E2 3850.153} C_VEL
LIN {X 0,Y 537.476,Z 970.266,A -85,B 0,C 180,E1 3853.904,E2 3853.904} C_VEL
LIN {X 0,Y 537.029,Z 986.445,A -85,B 0,C 180,E1 3857.422,E2 3857.422} C_VEL
LIN {X 0,Y 536.815,Z 999.718,A -85,B 0,C 180,E1 3861.513,E2 3861.513} C_VEL
LIN {X 0,Y 536.655,Z 1006.957,A -85,B 0,C 180,E1 3865.161,E2 3865.161} C_VEL
LIN {X 0,Y 536.67,Z 1010.087,A -85,B 0,C 180,E1 3868.389,E2 3868.389} C_VEL
LIN {X 0,Y 536.799,Z 1010.088,A -85,B 0,C 180,E1 3871.611,E2 3871.611} C_VEL
LIN {X 0,Y 536.765,Z 1005.756,A -85,B 0,C 180,E1 3875.647,E2 3875.647} C_VEL
LIN {X 0,Y 536.836,Z 996.304,A -85,B 0,C 180,E1 3879.71,E2 3879.71} C_VEL
LIN {X 0,Y 537.255,Z 980.764,A -85,B 0,C 180,E1 3883.936,E2 3883.936} C_VEL
LIN {X 0,Y 538.052,Z 959.666,A -85,B 0,C 180,E1 3887.969,E2 3887.969} C_VEL
LIN {X 0,Y 539.339,Z 933.551,A -85,B 0,C 180,E1 3891.675,E2 3891.675} C_VEL
LIN {X 0,Y 541.01,Z 903.284,A -85,B 0,C 180,E1 3894.942,E2 3894.942} C_VEL
LIN {X 0,Y 542.904,Z 869.543,A -85,B 0,C 180,E1 3897.699,E2 3897.699} C_VEL
LIN {X 0,Y 544.722,Z 834.373,A -85,B 0,C 180,E1 3899.823,E2 3899.823} C_VEL
LIN {X 0,Y 546.212,Z 797.663,A -85,B 0,C 180,E1 3901.376,E2 3901.376} C_VEL
LIN {X 0,Y 547.35,Z 760.643,A -85,B 0,C 180,E1 3902.336,E2 3902.336} C_VEL
LIN {X 0,Y 547.139,Z 708.805,A -85,B 0,C 180,E1 3903.171,E2 3903.171} C_VEL
LIN {X 0,Y 536.356,Z 685.03,A -85,B 0,C 180,E1 3904.373,E2 3904.373} C_VEL
LIN {X 0,Y 536.031,Z 685.03,A -85,B 0,C 180,E1 3910.529,E2 3910.529} C_VEL
LIN {X 0,Y 535.977,Z 685.03,A -85,B 0,C 180,E1 3917.055,E2 3917.055} C_VEL
LIN {X 0,Y 536.172,Z 685.03,A -85,B 0,C 180,E1 3922.001,E2 3922.001} C_VEL
LIN {X 0,Y 536.186,Z 685.03,A -85,B 0,C 180,E1 3927.674,E2 3927.674} C_VEL
LIN {X 0,Y 536.029,Z 685.03,A -85,B 0,C 180,E1 3933.228,E2 3933.228} C_VEL
LIN {X 0,Y 536.081,Z 685.03,A -85,B 0,C 180,E1 3938.533,E2 3938.533} C_VEL
LIN {X 0,Y 536.257,Z 685.03,A -85,B 0,C 180,E1 3943.655,E2 3943.655} C_VEL
LIN {X 0,Y 536.269,Z 685.03,A -85,B 0,C 180,E1 3948.638,E2 3948.638} C_VEL
LIN {X 0,Y 536.387,Z 685.03,A -85,B 0,C 180,E1 3953.536,E2 3953.536} C_VEL
LIN {X 0,Y 536.402,Z 685.03,A -85,B 0,C 180,E1 3958.385,E2 3958.385} C_VEL
LIN {X 0,Y 536.441,Z 685.03,A -85,B 0,C 180,E1 3963.222,E2 3963.222} C_VEL
LIN {X 0,Y 536.311,Z 685.03,A -85,B 0,C 180,E1 3968.084,E2 3968.084} C_VEL
LIN {X 0,Y 536.3,Z 685.03,A -85,B 0,C 180,E1 3973.004,E2 3973.004} C_VEL
LIN {X 0,Y 536.238,Z 685.03,A -85,B 0,C 180,E1 3978.027,E2 3978.027} C_VEL
LIN {X 0,Y 536.171,Z 685.03,A -85,B 0,C 180,E1 3983.199,E2 3983.199} C_VEL
LIN {X 0,Y 535.984,Z 685.03,A -85,B 0,C 180,E1 3989.219,E2 3989.219} C_VEL
LIN {X 0,Y 536.006,Z 685.03,A -85,B 0,C 180,E1 3995.272,E2 3995.272} C_VEL
LIN {X 0,Y 536.052,Z 685.03,A -85,B 0,C 180,E1 4000.531,E2 4000.531} C_VEL
LIN {X 0,Y 535.942,Z 685.03,A -85,B 0,C 180,E1 4005.26,E2 4005.26} C_VEL
LIN {X 0,Y 536.015,Z 685.03,A -85,B 0,C 180,E1 4011.732,E2 4011.732} C_VEL
LIN {X 0,Y 536.181,Z 685.03,A -85,B 0,C 180,E1 4017.675,E2 4017.675} C_VEL
LIN {X 0,Y 536.289,Z 685.03,A -85,B 0,C 180,E1 4022.8,E2 4022.8} C_VEL
LIN {X 0,Y 542.709,Z 710.2,A -85,B 0,C 180,E1 4024.327,E2 4024.327} C_VEL
LIN {X 0,Y 541.149,Z 744.574,A -85,B 0,C 180,E1 4026.478,E2 4026.478} C_VEL
LIN {X 0,Y 539.641,Z 775.063,A -85,B 0,C 180,E1 4029.119,E2 4029.119} C_VEL
LIN {X 0,Y 538.3,Z 802.862,A -85,B 0,C 180,E1 4032.361,E2 4032.361} C_VEL
LIN {X 0,Y 537.464,Z 824.588,A -85,B 0,C 180,E1 4035.809,E2 4035.809} C_VEL
LIN {X 0,Y 537.028,Z 841.461,A -85,B 0,C 180,E1 4039.526,E2 4039.526} C_VEL
LIN {X 0,Y 536.817,Z 851.506,A -85,B 0,C 180,E1 4042.733,E2 4042.733} C_VEL
LIN {X 0,Y 536.811,Z 858.727,A -85,B 0,C 180,E1 4046.777,E2 4046.777} C_VEL
LIN {X 0,Y 536.701,Z 860.497,A -85,B 0,C 180,E1 4050,E2 4050} C_VEL
LIN {X 0,Y 536.776,Z 857.636,A -85,B 0,C 180,E1 4054.022,E2 4054.022} C_VEL
LIN {X 0,Y 536.914,Z 849.059,A -85,B 0,C 180,E1 4058.078,E2 4058.078} C_VEL
LIN {X 0,Y 537.166,Z 835.965,A -85,B 0,C 180,E1 4061.751,E2 4061.751} C_VEL
LIN {X 0,Y 537.795,Z 816.835,A -85,B 0,C 180,E1 4065.46,E2 4065.46} C_VEL
LIN {X 0,Y 538.781,Z 793.165,A -85,B 0,C 180,E1 4068.789,E2 4068.789} C_VEL
LIN {X 0,Y 540.111,Z 765.314,A -85,B 0,C 180,E1 4071.724,E2 4071.724} C_VEL
LIN {X 0,Y 541.676,Z 732.8,A -85,B 0,C 180,E1 4074.262,E2 4074.262} C_VEL
LIN {X 0,Y 542.176,Z 704.935,A -85,B 0,C 180,E1 4075.884,E2 4075.884} C_VEL
LIN {X 0,Y 536.339,Z 685.03,A -85,B 0,C 180,E1 4077.16,E2 4077.16} C_VEL
LIN {X 0,Y 536.13,Z 685.03,A -85,B 0,C 180,E1 4082.407,E2 4082.407} C_VEL
LIN {X 0,Y 536.018,Z 685.03,A -85,B 0,C 180,E1 4088.268,E2 4088.268} C_VEL
LIN {X 0,Y 535.951,Z 685.03,A -85,B 0,C 180,E1 4094.74,E2 4094.74} C_VEL
LIN {X 0,Y 536.058,Z 685.03,A -85,B 0,C 180,E1 4099.658,E2 4099.658} C_VEL
LIN {X 0,Y 536.029,Z 685.03,A -85,B 0,C 180,E1 4104.725,E2 4104.725} C_VEL
LIN {X 0,Y 536.01,Z 685.03,A -85,B 0,C 180,E1 4110.776,E2 4110.776} C_VEL
LIN {X 0,Y 536.173,Z 685.03,A -85,B 0,C 180,E1 4116.801,E2 4116.801} C_VEL
LIN {X 0,Y 536.315,Z 685.03,A -85,B 0,C 180,E1 4121.976,E2 4121.976} C_VEL
LIN {X 0,Y 536.482,Z 685.03,A -85,B 0,C 180,E1 4127,E2 4127} C_VEL
LIN {X 0,Y 536.356,Z 685.03,A -85,B 0,C 180,E1 4132.65,E2 4132.65} C_VEL
LIN {X 0,Y 536.38,Z 685.03,A -85,B 0,C 180,E1 4138.391,E2 4138.391} C_VEL
LIN {X 0,Y 536.443,Z 685.03,A -85,B 0,C 180,E1 4143.228,E2 4143.228} C_VEL
LIN {X 0,Y 536.306,Z 685.03,A -85,B 0,C 180,E1 4148.09,E2 4148.09} C_VEL
LIN {X 0,Y 536.258,Z 685.03,A -85,B 0,C 180,E1 4153.012,E2 4153.012} C_VEL
LIN {X 0,Y 536.217,Z 685.03,A -85,B 0,C 180,E1 4158.034,E2 4158.034} C_VEL
LIN {X 0,Y 536.111,Z 685.03,A -85,B 0,C 180,E1 4163.209,E2 4163.209} C_VEL
LIN {X 0,Y 536.092,Z 685.03,A -85,B 0,C 180,E1 4166.76,E2 4166.76} C_VEL
LIN {X 0,Y 533.564,Z 685.03,A -85,B 0,C 180,E1 4168.14,E2 4168.14} C_VEL
LIN {X 0,Y 528.096,Z 685.03,A -85,B 0,C 180,E1 4170.207,E2 4170.207} C_VEL
LIN {X 0,Y 528.007,Z 685.03,A -85,B 0,C 180,E1 4170.446,E2 4170.446} C_VEL
LIN {X 0,Y 528.028,Z 685.03,A -85,B 0,C 180,E1 4176.88,E2 4176.88} C_VEL
LIN {X 0,Y 527.957,Z 685.03,A -85,B 0,C 180,E1 4183.312,E2 4183.312} C_VEL
LIN {X 0,Y 528.062,Z 685.03,A -85,B 0,C 180,E1 4188.91,E2 4188.91} C_VEL
LIN {X 0,Y 528.391,Z 685.063,A -85,B 0,C 180,E1 4195.105,E2 4195.105} C_VEL
LIN {X 0,Y 536.171,Z 702.133,A -85,B 0,C 180,E1 4195.953,E2 4195.953} C_VEL
LIN {X 0,Y 540.947,Z 714.125,A -85,B 0,C 180,E1 4196.482,E2 4196.482} C_VEL
LIN {X 0,Y 540.171,Z 776.993,A -85,B 0,C 180,E1 4197.564,E2 4197.564} C_VEL
LIN {X 0,Y 538.747,Z 815.401,A -85,B 0,C 180,E1 4198.858,E2 4198.858} C_VEL
LIN {X 0,Y 536.703,Z 853.663,A -85,B 0,C 180,E1 4200.838,E2 4200.838} C_VEL
LIN {X 0,Y 534.568,Z 888.659,A -85,B 0,C 180,E1 4203.377,E2 4203.377} C_VEL
LIN {X 0,Y 532.621,Z 920.039,A -85,B 0,C 180,E1 4206.411,E2 4206.411} C_VEL
LIN {X 0,Y 530.962,Z 947.121,A -85,B 0,C 180,E1 4209.824,E2 4209.824} C_VEL
LIN {X 0,Y 529.755,Z 970.268,A -85,B 0,C 180,E1 4213.663,E2 4213.663} C_VEL
LIN {X 0,Y 529.125,Z 987.983,A -85,B 0,C 180,E1 4217.65,E2 4217.65} C_VEL
LIN {X 0,Y 528.923,Z 999.718,A -85,B 0,C 180,E1 4221.386,E2 4221.386} C_VEL
LIN {X 0,Y 528.766,Z 1006.957,A -85,B 0,C 180,E1 4225.089,E2 4225.089} C_VEL
LIN {X 0,Y 528.768,Z 1010.088,A -85,B 0,C 180,E1 4228.365,E2 4228.365} C_VEL
LIN {X 0,Y 528.745,Z 1009.397,A -85,B 0,C 180,E1 4232.748,E2 4232.748} C_VEL
LIN {X 0,Y 528.86,Z 1004.223,A -85,B 0,C 180,E1 4236.554,E2 4236.554} C_VEL
LIN {X 0,Y 528.964,Z 994.369,A -85,B 0,C 180,E1 4240.489,E2 4240.489} C_VEL
LIN {X 0,Y 529.509,Z 979.148,A -85,B 0,C 180,E1 4244.503,E2 4244.503} C_VEL
LIN {X 0,Y 530.403,Z 958.343,A -85,B 0,C 180,E1 4248.452,E2 4248.452} C_VEL
LIN {X 0,Y 531.823,Z 932.641,A -85,B 0,C 180,E1 4252.112,E2 4252.112} C_VEL
LIN {X 0,Y 533.604,Z 903.613,A -85,B 0,C 180,E1 4255.28,E2 4255.28} C_VEL
LIN {X 0,Y 535.693,Z 870.386,A -85,B 0,C 180,E1 4258.041,E2 4258.041} C_VEL
LIN {X 0,Y 537.786,Z 834.151,A -85,B 0,C 180,E1 4260.259,E2 4260.259} C_VEL
LIN {X 0,Y 539.455,Z 797.659,A -85,B 0,C 180,E1 4261.814,E2 4261.814} C_VEL
LIN {X 0,Y 540.711,Z 759.329,A -85,B 0,C 180,E1 4262.806,E2 4262.806} C_VEL
LIN {X 0,Y 540.482,Z 711.234,A -85,B 0,C 180,E1 4263.596,E2 4263.596} C_VEL
LIN {X 0,Y 528.405,Z 685.03,A -85,B 0,C 180,E1 4264.958,E2 4264.958} C_VEL
LIN {X 0,Y 528.045,Z 685.03,A -85,B 0,C 180,E1 4271.092,E2 4271.092} C_VEL
LIN {X 0,Y 528.025,Z 685.03,A -85,B 0,C 180,E1 4276.695,E2 4276.695} C_VEL
LIN {X 0,Y 528.251,Z 685.03,A -85,B 0,C 180,E1 4283.138,E2 4283.138} C_VEL
LIN {X 0,Y 528.205,Z 685.03,A -85,B 0,C 180,E1 4288.987,E2 4288.987} C_VEL
LIN {X 0,Y 528.132,Z 685.03,A -85,B 0,C 180,E1 4294.621,E2 4294.621} C_VEL
LIN {X 0,Y 528.314,Z 685.03,A -85,B 0,C 180,E1 4300.486,E2 4300.486} C_VEL
LIN {X 0,Y 528.456,Z 685.03,A -85,B 0,C 180,E1 4306.793,E2 4306.793} C_VEL
LIN {X 0,Y 528.484,Z 685.03,A -85,B 0,C 180,E1 4311.79,E2 4311.79} C_VEL
LIN {X 0,Y 528.728,Z 685.03,A -85,B 0,C 180,E1 4316.725,E2 4316.725} C_VEL
LIN {X 0,Y 528.64,Z 685.03,A -85,B 0,C 180,E1 4322.475,E2 4322.475} C_VEL
LIN {X 0,Y 528.415,Z 685.03,A -85,B 0,C 180,E1 4328.205,E2 4328.205} C_VEL
LIN {X 0,Y 528.343,Z 685.03,A -85,B 0,C 180,E1 4333.816,E2 4333.816} C_VEL
LIN {X 0,Y 528.352,Z 685.03,A -85,B 0,C 180,E1 4339.526,E2 4339.526} C_VEL
LIN {X 0,Y 528.217,Z 685.03,A -85,B 0,C 180,E1 4345.368,E2 4345.368} C_VEL
LIN {X 0,Y 528.053,Z 685.03,A -85,B 0,C 180,E1 4350.986,E2 4350.986} C_VEL
LIN {X 0,Y 528.165,Z 685.03,A -85,B 0,C 180,E1 4356.873,E2 4356.873} C_VEL
LIN {X 0,Y 528.061,Z 685.03,A -85,B 0,C 180,E1 4363.292,E2 4363.292} C_VEL
LIN {X 0,Y 527.966,Z 685.03,A -85,B 0,C 180,E1 4368.901,E2 4368.901} C_VEL
LIN {X 0,Y 528.16,Z 685.03,A -85,B 0,C 180,E1 4375.151,E2 4375.151} C_VEL
LIN {X 0,Y 528.307,Z 685.03,A -85,B 0,C 180,E1 4380.95,E2 4380.95} C_VEL
LIN {X 0,Y 528.401,Z 685.432,A -85,B 0,C 180,E1 4382.378,E2 4382.378} C_VEL
LIN {X 0,Y 535.501,Z 710.783,A -85,B 0,C 180,E1 4383.987,E2 4383.987} C_VEL
LIN {X 0,Y 533.775,Z 744.561,A -85,B 0,C 180,E1 4386.133,E2 4386.133} C_VEL
LIN {X 0,Y 532.086,Z 775.378,A -85,B 0,C 180,E1 4388.842,E2 4388.842} C_VEL
LIN {X 0,Y 530.613,Z 802.857,A -85,B 0,C 180,E1 4392.097,E2 4392.097} C_VEL
LIN {X 0,Y 529.648,Z 824.573,A -85,B 0,C 180,E1 4395.593,E2 4395.593} C_VEL
LIN {X 0,Y 529.143,Z 841.458,A -85,B 0,C 180,E1 4399.368,E2 4399.368} C_VEL
LIN {X 0,Y 528.923,Z 851.504,A -85,B 0,C 180,E1 4402.624,E2 4402.624} C_VEL
LIN {X 0,Y 528.915,Z 858.779,A -85,B 0,C 180,E1 4406.779,E2 4406.779} C_VEL
LIN {X 0,Y 528.801,Z 860.497,A -85,B 0,C 180,E1 4410,E2 4410} C_VEL
LIN {X 0,Y 528.873,Z 857.625,A -85,B 0,C 180,E1 4414.09,E2 4414.09} C_VEL
LIN {X 0,Y 529.036,Z 849.061,A -85,B 0,C 180,E1 4418.199,E2 4418.199} C_VEL
LIN {X 0,Y 529.306,Z 835.969,A -85,B 0,C 180,E1 4421.928,E2 4421.928} C_VEL
LIN {X 0,Y 530.003,Z 816.839,A -85,B 0,C 180,E1 4425.693,E2 4425.693} C_VEL
LIN {X 0,Y 531.159,Z 793.17,A -85,B 0,C 180,E1 4429.069,E2 4429.069} C_VEL
LIN {X 0,Y 532.654,Z 764.831,A -85,B 0,C 180,E1 4432.091,E2 4432.091} C_VEL
LIN {X 0,Y 534.386,Z 732.812,A -85,B 0,C 180,E1 4434.614,E2 4434.614} C_VEL
LIN {X 0,Y 534.766,Z 706.63,A -85,B 0,C 180,E1 4436.18,E2 4436.18} C_VEL
LIN {X 0,Y 528.392,Z 685.03,A -85,B 0,C 180,E1 4437.649,E2 4437.649} C_VEL
LIN {X 0,Y 528.188,Z 685.03,A -85,B 0,C 180,E1 4444.066,E2 4444.066} C_VEL
LIN {X 0,Y 527.991,Z 685.03,A -85,B 0,C 180,E1 4449.507,E2 4449.507} C_VEL
LIN {X 0,Y 528.064,Z 685.03,A -85,B 0,C 180,E1 4455.594,E2 4455.594} C_VEL
LIN {X 0,Y 528.125,Z 685.03,A -85,B 0,C 180,E1 4461.061,E2 4461.061} C_VEL
LIN {X 0,Y 528.101,Z 685.03,A -85,B 0,C 180,E1 4467.125,E2 4467.125} C_VEL
LIN {X 0,Y 528.149,Z 685.03,A -85,B 0,C 180,E1 4472.803,E2 4472.803} C_VEL
LIN {X 0,Y 528.315,Z 685.03,A -85,B 0,C 180,E1 4478.209,E2 4478.209} C_VEL
LIN {X 0,Y 528.443,Z 685.03,A -85,B 0,C 180,E1 4483.413,E2 4483.413} C_VEL
LIN {X 0,Y 528.461,Z 685.03,A -85,B 0,C 180,E1 4488.474,E2 4488.474} C_VEL
LIN {X 0,Y 528.503,Z 685.03,A -85,B 0,C 180,E1 4493.446,E2 4493.446} C_VEL
LIN {X 0,Y 528.481,Z 685.03,A -85,B 0,C 180,E1 4498.367,E2 4498.367} C_VEL
LIN {X 0,Y 528.558,Z 685.03,A -85,B 0,C 180,E1 4503.276,E2 4503.276} C_VEL
LIN {X 0,Y 528.41,Z 685.03,A -85,B 0,C 180,E1 4508.212,E2 4508.212} C_VEL
LIN {X 0,Y 528.315,Z 685.03,A -85,B 0,C 180,E1 4513.804,E2 4513.804} C_VEL
LIN {X 0,Y 528.298,Z 685.03,A -85,B 0,C 180,E1 4519.509,E2 4519.509} C_VEL
LIN {X 0,Y 528.199,Z 685.03,A -85,B 0,C 180,E1 4525.376,E2 4525.376} C_VEL
LIN {X 0,Y 528.007,Z 685.03,A -85,B 0,C 180,E1 4530.446,E2 4530.446} C_VEL
LIN {X 0,Y 525.502,Z 685.03,A -85,B 0,C 180,E1 4531.849,E2 4531.849} C_VEL
LIN {X 0,Y 520.103,Z 685.03,A -85,B 0,C 180,E1 4533.95,E2 4533.95} C_VEL
LIN {X 0,Y 519.996,Z 685.03,A -85,B 0,C 180,E1 4534.193,E2 4534.193} C_VEL
LIN {X 0,Y 520.04,Z 685.03,A -85,B 0,C 180,E1 4539.671,E2 4539.671} C_VEL
LIN {X 0,Y 520.083,Z 685.03,A -85,B 0,C 180,E1 4545.865,E2 4545.865} C_VEL
LIN {X 0,Y 520.232,Z 685.03,A -85,B 0,C 180,E1 4551.551,E2 4551.551} C_VEL
LIN {X 0,Y 520.451,Z 685.258,A -85,B 0,C 180,E1 4554.5,E2 4554.5} C_VEL
LIN {X 0,Y 534.362,Z 716.407,A -85,B 0,C 180,E1 4556.049,E2 4556.049} C_VEL
LIN {X 0,Y 533.512,Z 776.992,A -85,B 0,C 180,E1 4557.108,E2 4557.108} C_VEL
LIN {X 0,Y 531.902,Z 815.763,A -85,B 0,C 180,E1 4558.428,E2 4558.428} C_VEL
LIN {X 0,Y 529.704,Z 853.66,A -85,B 0,C 180,E1 4560.415,E2 4560.415} C_VEL
LIN {X 0,Y 527.329,Z 888.654,A -85,B 0,C 180,E1 4562.982,E2 4562.982} C_VEL
LIN {X 0,Y 525.145,Z 920.161,A -85,B 0,C 180,E1 4566.068,E2 4566.068} C_VEL
LIN {X 0,Y 523.322,Z 947.397,A -85,B 0,C 180,E1 4569.558,E2 4569.558} C_VEL
LIN {X 0,Y 521.987,Z 970.269,A -85,B 0,C 180,E1 4573.413,E2 4573.413} C_VEL
LIN {X 0,Y 521.281,Z 987.984,A -85,B 0,C 180,E1 4577.461,E2 4577.461} C_VEL
LIN {X 0,Y 521.053,Z 999.718,A -85,B 0,C 180,E1 4581.255,E2 4581.255} C_VEL
LIN {X 0,Y 520.871,Z 1006.957,A -85,B 0,C 180,E1 4585.014,E2 4585.014} C_VEL
LIN {X 0,Y 520.882,Z 1010.088,A -85,B 0,C 180,E1 4588.34,E2 4588.34} C_VEL
LIN {X 0,Y 520.996,Z 1010.088,A -85,B 0,C 180,E1 4591.66,E2 4591.66} C_VEL
LIN {X 0,Y 521.001,Z 1005.755,A -85,B 0,C 180,E1 4595.818,E2 4595.818} C_VEL
LIN {X 0,Y 521.079,Z 996.125,A -85,B 0,C 180,E1 4600.072,E2 4600.072} C_VEL
LIN {X 0,Y 521.601,Z 981.261,A -85,B 0,C 180,E1 4604.241,E2 4604.241} C_VEL
LIN {X 0,Y 522.633,Z 959.663,A -85,B 0,C 180,E1 4608.518,E2 4608.518} C_VEL
LIN {X 0,Y 524.234,Z 933.289,A -85,B 0,C 180,E1 4612.366,E2 4612.366} C_VEL
LIN {X 0,Y 526.296,Z 903.173,A -85,B 0,C 180,E1 4615.7,E2 4615.7} C_VEL
LIN {X 0,Y 528.591,Z 869.761,A -85,B 0,C 180,E1 4618.499,E2 4618.499} C_VEL
LIN {X 0,Y 530.883,Z 833.878,A -85,B 0,C 180,E1 4620.71,E2 4620.71} C_VEL
LIN {X 0,Y 532.686,Z 797.462,A -85,B 0,C 180,E1 4622.274,E2 4622.274} C_VEL
LIN {X 0,Y 534.081,Z 760.072,A -85,B 0,C 180,E1 4623.252,E2 4623.252} C_VEL
LIN {X 0,Y 533.71,Z 713.467,A -85,B 0,C 180,E1 4624.045,E2 4624.045} C_VEL
LIN {X 0,Y 520.474,Z 685.03,A -85,B 0,C 180,E1 4625.567,E2 4625.567} C_VEL
LIN {X 0,Y 520.112,Z 685.03,A -85,B 0,C 180,E1 4631.859,E2 4631.859} C_VEL
LIN {X 0,Y 520.147,Z 685.03,A -85,B 0,C 180,E1 4638.144,E2 4638.144} C_VEL
LIN {X 0,Y 520.326,Z 685.03,A -85,B 0,C 180,E1 4644.294,E2 4644.294} C_VEL
LIN {X 0,Y 520.293,Z 685.03,A -85,B 0,C 180,E1 4648.529,E2 4648.529} C_VEL
LIN {X 0,Y 520.175,Z 685.03,A -85,B 0,C 180,E1 4654.204,E2 4654.204} C_VEL
LIN {X 0,Y 520.304,Z 685.03,A -85,B 0,C 180,E1 4659.632,E2 4659.632} C_VEL
LIN {X 0,Y 520.489,Z 685.03,A -85,B 0,C 180,E1 4664.873,E2 4664.873} C_VEL
LIN {X 0,Y 520.541,Z 685.03,A -85,B 0,C 180,E1 4670.272,E2 4670.272} C_VEL
LIN {X 0,Y 520.817,Z 685.03,A -85,B 0,C 180,E1 4676.675,E2 4676.675} C_VEL
LIN {X 0,Y 520.907,Z 685.03,A -85,B 0,C 180,E1 4681.657,E2 4681.657} C_VEL
LIN {X 0,Y 520.717,Z 685.03,A -85,B 0,C 180,E1 4686.653,E2 4686.653} C_VEL
LIN {X 0,Y 520.533,Z 685.03,A -85,B 0,C 180,E1 4691.704,E2 4691.704} C_VEL
LIN {X 0,Y 520.427,Z 685.03,A -85,B 0,C 180,E1 4696.894,E2 4696.894} C_VEL
LIN {X 0,Y 520.366,Z 685.03,A -85,B 0,C 180,E1 4702.142,E2 4702.142} C_VEL
LIN {X 0,Y 520.224,Z 685.03,A -85,B 0,C 180,E1 4707.647,E2 4707.647} C_VEL
LIN {X 0,Y 520.116,Z 685.03,A -85,B 0,C 180,E1 4713.445,E2 4713.445} C_VEL
LIN {X 0,Y 520.222,Z 685.03,A -85,B 0,C 180,E1 4719.646,E2 4719.646} C_VEL
LIN {X 0,Y 520.097,Z 685.03,A -85,B 0,C 180,E1 4725.867,E2 4725.867} C_VEL
LIN {X 0,Y 520.087,Z 685.03,A -85,B 0,C 180,E1 4731.561,E2 4731.561} C_VEL
LIN {X 0,Y 520.346,Z 685.03,A -85,B 0,C 180,E1 4737.233,E2 4737.233} C_VEL
LIN {X 0,Y 520.431,Z 685.309,A -85,B 0,C 180,E1 4741.777,E2 4741.777} C_VEL
LIN {X 0,Y 528.186,Z 713.356,A -85,B 0,C 180,E1 4743.748,E2 4743.748} C_VEL
LIN {X 0,Y 526.359,Z 745.938,A -85,B 0,C 180,E1 4745.888,E2 4745.888} C_VEL
LIN {X 0,Y 524.535,Z 776.083,A -85,B 0,C 180,E1 4748.598,E2 4748.598} C_VEL
LIN {X 0,Y 522.979,Z 802.315,A -85,B 0,C 180,E1 4751.752,E2 4751.752} C_VEL
LIN {X 0,Y 521.911,Z 823.787,A -85,B 0,C 180,E1 4755.22,E2 4755.22} C_VEL
LIN {X 0,Y 521.274,Z 839.706,A -85,B 0,C 180,E1 4758.723,E2 4758.723} C_VEL
LIN {X 0,Y 521.043,Z 851.502,A -85,B 0,C 180,E1 4762.512,E2 4762.512} C_VEL
LIN {X 0,Y 521.001,Z 858.725,A -85,B 0,C 180,E1 4766.679,E2 4766.679} C_VEL
LIN {X 0,Y 520.906,Z 860.497,A -85,B 0,C 180,E1 4770,E2 4770} C_VEL
LIN {X 0,Y 520.971,Z 857.626,A -85,B 0,C 180,E1 4774.153,E2 4774.153} C_VEL
LIN {X 0,Y 521.153,Z 849.063,A -85,B 0,C 180,E1 4778.324,E2 4778.324} C_VEL
LIN {X 0,Y 521.477,Z 835.973,A -85,B 0,C 180,E1 4782.11,E2 4782.11} C_VEL
LIN {X 0,Y 522.223,Z 816.843,A -85,B 0,C 180,E1 4785.933,E2 4785.933} C_VEL
LIN {X 0,Y 523.535,Z 793.175,A -85,B 0,C 180,E1 4789.358,E2 4789.358} C_VEL
LIN {X 0,Y 525.112,Z 766.194,A -85,B 0,C 180,E1 4792.293,E2 4792.293} C_VEL
LIN {X 0,Y 527.012,Z 734.366,A -85,B 0,C 180,E1 4794.869,E2 4794.869} C_VEL
LIN {X 0,Y 527.532,Z 708.862,A -85,B 0,C 180,E1 4796.448,E2 4796.448} C_VEL
LIN {X 0,Y 520.403,Z 685.03,A -85,B 0,C 180,E1 4798.185,E2 4798.185} C_VEL
LIN {X 0,Y 520.261,Z 685.03,A -85,B 0,C 180,E1 4803.442,E2 4803.442} C_VEL
LIN {X 0,Y 520.1,Z 685.03,A -85,B 0,C 180,E1 4809.665,E2 4809.665} C_VEL
LIN {X 0,Y 520.146,Z 685.03,A -85,B 0,C 180,E1 4815.881,E2 4815.881} C_VEL
LIN {X 0,Y 520.196,Z 685.03,A -85,B 0,C 180,E1 4821.556,E2 4821.556} C_VEL
LIN {X 0,Y 520.183,Z 685.03,A -85,B 0,C 180,E1 4827.273,E2 4827.273} C_VEL
LIN {X 0,Y 520.247,Z 685.03,A -85,B 0,C 180,E1 4832.355,E2 4832.355} C_VEL
LIN {X 0,Y 520.397,Z 685.03,A -85,B 0,C 180,E1 4838.11,E2 4838.11} C_VEL
LIN {X 0,Y 520.516,Z 685.03,A -85,B 0,C 180,E1 4843.152,E2 4843.152} C_VEL
LIN {X 0,Y 520.562,Z 685.03,A -85,B 0,C 180,E1 4848.297,E2 4848.297} C_VEL
LIN {X 0,Y 520.591,Z 685.03,A -85,B 0,C 180,E1 4853.346,E2 4853.346} C_VEL
LIN {X 0,Y 520.608,Z 685.03,A -85,B 0,C 180,E1 4858.342,E2 4858.342} C_VEL
LIN {X 0,Y 520.652,Z 685.03,A -85,B 0,C 180,E1 4863.326,E2 4863.326} C_VEL
LIN {X 0,Y 520.499,Z 685.03,A -85,B 0,C 180,E1 4868.337,E2 4868.337} C_VEL
LIN {X 0,Y 520.453,Z 685.03,A -85,B 0,C 180,E1 4873.414,E2 4873.414} C_VEL
LIN {X 0,Y 520.385,Z 685.03,A -85,B 0,C 180,E1 4878.603,E2 4878.603} C_VEL
LIN {X 0,Y 520.27,Z 685.03,A -85,B 0,C 180,E1 4883.959,E2 4883.959} C_VEL
LIN {X 0,Y 520.168,Z 685.03,A -85,B 0,C 180,E1 4889.55,E2 4889.55} C_VEL
LIN {X 0,Y 519.996,Z 685.03,A -85,B 0,C 180,E1 4894.193,E2 4894.193} C_VEL
LIN {X 0,Y 515.995,Z 685.03,A -85,B 0,C 180,E1 4896.078,E2 4896.078} C_VEL
